LIN {X 0,Y 574.016,Z 518.024,A -85,B 0,C 180,E1 -2272.305,E2 -2272.305} C_VEL
LIN {X 0,Y 573.235,Z 513.083,A -85,B 0,C 180,E1 -2273.099,E2 -2273.099} C_VEL
LIN {X 0,Y 573.254,Z 513.082,A -85,B 0,C 180,E1 -2275.409,E2 -2275.409} C_VEL
LIN {X 0,Y 573.253,Z 513.075,A -85,B 0,C 180,E1 -2278.029,E2 -2278.029} C_VEL
LIN {X 0,Y 573.238,Z 513.077,A -85,B 0,C 180,E1 -2280.883,E2 -2280.883} C_VEL
LIN {X 0,Y 573.261,Z 513.081,A -85,B 0,C 180,E1 -2283.523,E2 -2283.523} C_VEL
LIN {X 0,Y 573.236,Z 513.076,A -85,B 0,C 180,E1 -2286.049,E2 -2286.049} C_VEL
LIN {X 0,Y 573.246,Z 513.073,A -85,B 0,C 180,E1 -2288.7,E2 -2288.7} C_VEL
LIN {X 0,Y 573.251,Z 513.08,A -85,B 0,C 180,E1 -2291.595,E2 -2291.595} C_VEL
LIN {X 0,Y 573.235,Z 513.074,A -85,B 0,C 180,E1 -2294.332,E2 -2294.332} C_VEL
LIN {X 0,Y 573.234,Z 513.083,A -85,B 0,C 180,E1 -2297.358,E2 -2297.358} C_VEL
LIN {X 0,Y 573.243,Z 513.073,A -85,B 0,C 180,E1 -2300.392,E2 -2300.392} C_VEL
LIN {X 0,Y 573.25,Z 513.077,A -85,B 0,C 180,E1 -2303.077,E2 -2303.077} C_VEL
LIN {X 0,Y 573.269,Z 513.077,A -85,B 0,C 180,E1 -2305.671,E2 -2305.671} C_VEL
LIN {X 0,Y 573.243,Z 513.074,A -85,B 0,C 180,E1 -2308.185,E2 -2308.185} C_VEL
LIN {X 0,Y 573.263,Z 513.071,A -85,B 0,C 180,E1 -2310.634,E2 -2310.634} C_VEL
LIN {X 0,Y 573.262,Z 513.081,A -85,B 0,C 180,E1 -2313.5,E2 -2313.5} C_VEL
LIN {X 0,Y 573.224,Z 513.077,A -85,B 0,C 180,E1 -2316.134,E2 -2316.134} C_VEL
LIN {X 0,Y 573.253,Z 513.078,A -85,B 0,C 180,E1 -2319.174,E2 -2319.174} C_VEL
LIN {X 0,Y 573.232,Z 513.085,A -85,B 0,C 180,E1 -2321.412,E2 -2321.412} C_VEL
LIN {X 0,Y 573.249,Z 513.08,A -85,B 0,C 180,E1 -2323.622,E2 -2323.622} C_VEL
LIN {X 0,Y 573.227,Z 513.075,A -85,B 0,C 180,E1 -2326.529,E2 -2326.529} C_VEL
LIN {X 0,Y 573.273,Z 513.07,A -85,B 0,C 180,E1 -2328.734,E2 -2328.734} C_VEL
LIN {X 0,Y 573.298,Z 513.075,A -85,B 0,C 180,E1 -2331.541,E2 -2331.541} C_VEL
LIN {X 0,Y 573.283,Z 513.068,A -85,B 0,C 180,E1 -2334.372,E2 -2334.372} C_VEL
LIN {X 0,Y 573.3,Z 513.069,A -85,B 0,C 180,E1 -2337.892,E2 -2337.892} C_VEL
LIN {X 0,Y 573.328,Z 513.063,A -85,B 0,C 180,E1 -2340.702,E2 -2340.702} C_VEL
LIN {X 0,Y 573.234,Z 513.083,A -85,B 0,C 180,E1 -2343.515,E2 -2343.515} C_VEL
LIN {X 0,Y 573.283,Z 513.075,A -85,B 0,C 180,E1 -2345.628,E2 -2345.628} C_VEL
LIN {X 0,Y 573.298,Z 513.066,A -85,B 0,C 180,E1 -2348.459,E2 -2348.459} C_VEL
LIN {X 0,Y 573.289,Z 513.076,A -85,B 0,C 180,E1 -2351.312,E2 -2351.312} C_VEL
LIN {X 0,Y 573.271,Z 513.07,A -85,B 0,C 180,E1 -2354.425,E2 -2354.425} C_VEL
LIN {X 0,Y 573.25,Z 513.077,A -85,B 0,C 180,E1 -2357.112,E2 -2357.112} C_VEL
LIN {X 0,Y 573.248,Z 513.074,A -85,B 0,C 180,E1 -2360.077,E2 -2360.077} C_VEL
LIN {X 0,Y 573.231,Z 513.075,A -85,B 0,C 180,E1 -2362.338,E2 -2362.338} C_VEL
LIN {X 0,Y 573.243,Z 513.073,A -85,B 0,C 180,E1 -2364.401,E2 -2364.401} C_VEL
LIN {X 0,Y 572.618,Z 513.155,A -85,B 0,C 180,E1 -2364.987,E2 -2364.987} C_VEL
LIN {X 0,Y 569.781,Z 513.514,A -85,B 0,C 180,E1 -2365.939,E2 -2365.939} C_VEL
LIN {X 0,Y 567.353,Z 513.82,A -85,B 0,C 180,E1 -2366.705,E2 -2366.705} C_VEL
LIN {X 0,Y 566.3,Z 513.947,A -85,B 0,C 180,E1 -2367.296,E2 -2367.296} C_VEL
LIN {X 0,Y 566.211,Z 513.956,A -85,B 0,C 180,E1 -2367.496,E2 -2367.496} C_VEL
LIN {X 0,Y 566.221,Z 513.953,A -85,B 0,C 180,E1 -2369.768,E2 -2369.768} C_VEL
LIN {X 0,Y 566.202,Z 513.95,A -85,B 0,C 180,E1 -2372.432,E2 -2372.432} C_VEL
LIN {X 0,Y 566.21,Z 513.953,A -85,B 0,C 180,E1 -2374.996,E2 -2374.996} C_VEL
LIN {X 0,Y 566.191,Z 513.961,A -85,B 0,C 180,E1 -2377.462,E2 -2377.462} C_VEL
LIN {X 0,Y 566.222,Z 513.948,A -85,B 0,C 180,E1 -2380.198,E2 -2380.198} C_VEL
LIN {X 0,Y 566.197,Z 513.956,A -85,B 0,C 180,E1 -2383.055,E2 -2383.055} C_VEL
LIN {X 0,Y 566.2,Z 513.952,A -85,B 0,C 180,E1 -2386.049,E2 -2386.049} C_VEL
LIN {X 0,Y 566.21,Z 513.952,A -85,B 0,C 180,E1 -2388.865,E2 -2388.865} C_VEL
LIN {X 0,Y 566.189,Z 513.958,A -85,B 0,C 180,E1 -2391.638,E2 -2391.638} C_VEL
LIN {X 0,Y 566.193,Z 513.952,A -85,B 0,C 180,E1 -2394.311,E2 -2394.311} C_VEL
LIN {X 0,Y 566.22,Z 513.951,A -85,B 0,C 180,E1 -2396.899,E2 -2396.899} C_VEL
LIN {X 0,Y 566.186,Z 513.963,A -85,B 0,C 180,E1 -2399.408,E2 -2399.408} C_VEL
LIN {X 0,Y 566.213,Z 513.952,A -85,B 0,C 180,E1 -2401.858,E2 -2401.858} C_VEL
LIN {X 0,Y 566.215,Z 513.949,A -85,B 0,C 180,E1 -2404.252,E2 -2404.252} C_VEL
LIN {X 0,Y 566.172,Z 513.955,A -85,B 0,C 180,E1 -2406.72,E2 -2406.72} C_VEL
LIN {X 0,Y 566.217,Z 513.956,A -85,B 0,C 180,E1 -2409.663,E2 -2409.663} C_VEL
LIN {X 0,Y 566.204,Z 513.953,A -85,B 0,C 180,E1 -2412.669,E2 -2412.669} C_VEL
LIN {X 0,Y 566.279,Z 514.062,A -85,B 0,C 180,E1 -2414.178,E2 -2414.178} C_VEL
LIN {X 0,Y 566.581,Z 518.022,A -85,B 0,C 180,E1 -2414.901,E2 -2414.901} C_VEL
LIN {X 0,Y 566.388,Z 534.477,A -85,B 0,C 180,E1 -2417.823,E2 -2417.823} C_VEL
LIN {X 0,Y 566.243,Z 547.118,A -85,B 0,C 180,E1 -2420.039,E2 -2420.039} C_VEL
LIN {X 0,Y 567.168,Z 552.643,A -85,B 0,C 180,E1 -2420.145,E2 -2420.145} C_VEL
LIN {X 0,Y 566.949,Z 653.825,A -85,B 0,C 180,E1 -2421.445,E2 -2421.445} C_VEL
LIN {X 0,Y 566.838,Z 667.023,A -85,B 0,C 180,E1 -2421.758,E2 -2421.758} C_VEL
LIN {X 0,Y 566.748,Z 679.661,A -85,B 0,C 180,E1 -2422.205,E2 -2422.205} C_VEL
LIN {X 0,Y 566.617,Z 691.734,A -85,B 0,C 180,E1 -2422.786,E2 -2422.786} C_VEL
LIN {X 0,Y 566.435,Z 703.285,A -85,B 0,C 180,E1 -2423.506,E2 -2423.506} C_VEL
LIN {X 0,Y 566.299,Z 714.55,A -85,B 0,C 180,E1 -2424.392,E2 -2424.392} C_VEL
LIN {X 0,Y 566.217,Z 724.449,A -85,B 0,C 180,E1 -2425.372,E2 -2425.372} C_VEL
LIN {X 0,Y 566.049,Z 733.188,A -85,B 0,C 180,E1 -2426.441,E2 -2426.441} C_VEL
LIN {X 0,Y 566.022,Z 740.193,A -85,B 0,C 180,E1 -2427.509,E2 -2427.509} C_VEL
LIN {X 0,Y 565.892,Z 745.807,A -85,B 0,C 180,E1 -2428.577,E2 -2428.577} C_VEL
LIN {X 0,Y 565.948,Z 750.233,A -85,B 0,C 180,E1 -2429.644,E2 -2429.644} C_VEL
LIN {X 0,Y 565.846,Z 753.603,A -85,B 0,C 180,E1 -2430.712,E2 -2430.712} C_VEL
LIN {X 0,Y 565.847,Z 755.279,A -85,B 0,C 180,E1 -2431.423,E2 -2431.423} C_VEL
LIN {X 0,Y 565.873,Z 757.434,A -85,B 0,C 180,E1 -2432.847,E2 -2432.847} C_VEL
LIN {X 0,Y 565.911,Z 757.899,A -85,B 0,C 180,E1 -2433.56,E2 -2433.56} C_VEL
LIN {X 0,Y 565.911,Z 757.956,A -85,B 0,C 180,E1 -2434.273,E2 -2434.273} C_VEL
LIN {X 0,Y 565.899,Z 756.923,A -85,B 0,C 180,E1 -2435.702,E2 -2435.702} C_VEL
LIN {X 0,Y 565.919,Z 755.545,A -85,B 0,C 180,E1 -2436.534,E2 -2436.534} C_VEL
LIN {X 0,Y 565.903,Z 752.224,A -85,B 0,C 180,E1 -2437.852,E2 -2437.852} C_VEL
LIN {X 0,Y 565.93,Z 748.356,A -85,B 0,C 180,E1 -2438.93,E2 -2438.93} C_VEL
LIN {X 0,Y 565.978,Z 743.338,A -85,B 0,C 180,E1 -2440.011,E2 -2440.011} C_VEL
LIN {X 0,Y 566.048,Z 736.125,A -85,B 0,C 180,E1 -2441.227,E2 -2441.227} C_VEL
LIN {X 0,Y 566.156,Z 727.551,A -85,B 0,C 180,E1 -2442.364,E2 -2442.364} C_VEL
LIN {X 0,Y 566.247,Z 719.111,A -85,B 0,C 180,E1 -2443.274,E2 -2443.274} C_VEL
LIN {X 0,Y 566.393,Z 708.668,A -85,B 0,C 180,E1 -2444.185,E2 -2444.185} C_VEL
LIN {X 0,Y 566.497,Z 697.979,A -85,B 0,C 180,E1 -2444.936,E2 -2444.936} C_VEL
LIN {X 0,Y 566.671,Z 686.887,A -85,B 0,C 180,E1 -2445.557,E2 -2445.557} C_VEL
LIN {X 0,Y 566.777,Z 675.235,A -85,B 0,C 180,E1 -2446.061,E2 -2446.061} C_VEL
LIN {X 0,Y 566.899,Z 662.692,A -85,B 0,C 180,E1 -2446.451,E2 -2446.451} C_VEL
LIN {X 0,Y 566.964,Z 650.026,A -85,B 0,C 180,E1 -2446.704,E2 -2446.704} C_VEL
LIN {X 0,Y 567.069,Z 552.012,A -85,B 0,C 180,E1 -2447.955,E2 -2447.955} C_VEL
LIN {X 0,Y 566.284,Z 547.177,A -85,B 0,C 180,E1 -2448.04,E2 -2448.04} C_VEL
LIN {X 0,Y 566.438,Z 529.829,A -85,B 0,C 180,E1 -2451.088,E2 -2451.088} C_VEL
LIN {X 0,Y 566.502,Z 515.841,A -85,B 0,C 180,E1 -2453.583,E2 -2453.583} C_VEL
LIN {X 0,Y 566.223,Z 513.955,A -85,B 0,C 180,E1 -2453.936,E2 -2453.936} C_VEL
LIN {X 0,Y 566.21,Z 513.96,A -85,B 0,C 180,E1 -2456.659,E2 -2456.659} C_VEL
LIN {X 0,Y 566.194,Z 513.959,A -85,B 0,C 180,E1 -2458.952,E2 -2458.952} C_VEL
LIN {X 0,Y 566.198,Z 513.952,A -85,B 0,C 180,E1 -2461.421,E2 -2461.421} C_VEL
LIN {X 0,Y 566.21,Z 513.951,A -85,B 0,C 180,E1 -2463.955,E2 -2463.955} C_VEL
LIN {X 0,Y 566.211,Z 513.958,A -85,B 0,C 180,E1 -2466.568,E2 -2466.568} C_VEL
LIN {X 0,Y 566.211,Z 513.95,A -85,B 0,C 180,E1 -2469.685,E2 -2469.685} C_VEL
LIN {X 0,Y 566.214,Z 513.951,A -85,B 0,C 180,E1 -2472.086,E2 -2472.086} C_VEL
LIN {X 0,Y 566.17,Z 513.959,A -85,B 0,C 180,E1 -2475.035,E2 -2475.035} C_VEL
LIN {X 0,Y 566.214,Z 513.951,A -85,B 0,C 180,E1 -2478.135,E2 -2478.135} C_VEL
LIN {X 0,Y 566.217,Z 513.958,A -85,B 0,C 180,E1 -2480.726,E2 -2480.726} C_VEL
LIN {X 0,Y 566.213,Z 513.949,A -85,B 0,C 180,E1 -2483.782,E2 -2483.782} C_VEL
LIN {X 0,Y 566.223,Z 513.952,A -85,B 0,C 180,E1 -2486.262,E2 -2486.262} C_VEL
LIN {X 0,Y 566.196,Z 513.956,A -85,B 0,C 180,E1 -2488.921,E2 -2488.921} C_VEL
LIN {X 0,Y 566.19,Z 513.956,A -85,B 0,C 180,E1 -2491.046,E2 -2491.046} C_VEL
LIN {X 0,Y 566.238,Z 513.945,A -85,B 0,C 180,E1 -2493.46,E2 -2493.46} C_VEL
LIN {X 0,Y 566.191,Z 513.952,A -85,B 0,C 180,E1 -2495.819,E2 -2495.819} C_VEL
LIN {X 0,Y 566.209,Z 513.956,A -85,B 0,C 180,E1 -2498.902,E2 -2498.902} C_VEL
LIN {X 0,Y 566.205,Z 513.952,A -85,B 0,C 180,E1 -2501.172,E2 -2501.172} C_VEL
LIN {X 0,Y 566.212,Z 513.95,A -85,B 0,C 180,E1 -2503.412,E2 -2503.412} C_VEL
LIN {X 0,Y 566.191,Z 513.957,A -85,B 0,C 180,E1 -2506.359,E2 -2506.359} C_VEL
LIN {X 0,Y 566.265,Z 513.953,A -85,B 0,C 180,E1 -2508.654,E2 -2508.654} C_VEL
LIN {X 0,Y 566.239,Z 513.946,A -85,B 0,C 180,E1 -2511.434,E2 -2511.434} C_VEL
LIN {X 0,Y 566.252,Z 513.949,A -85,B 0,C 180,E1 -2514.302,E2 -2514.302} C_VEL
LIN {X 0,Y 566.272,Z 513.941,A -85,B 0,C 180,E1 -2517.866,E2 -2517.866} C_VEL
LIN {X 0,Y 566.298,Z 513.947,A -85,B 0,C 180,E1 -2520.711,E2 -2520.711} C_VEL
LIN {X 0,Y 566.272,Z 513.947,A -85,B 0,C 180,E1 -2522.845,E2 -2522.845} C_VEL
LIN {X 0,Y 566.252,Z 513.945,A -85,B 0,C 180,E1 -2525.698,E2 -2525.698} C_VEL
LIN {X 0,Y 566.24,Z 513.955,A -85,B 0,C 180,E1 -2528.565,E2 -2528.565} C_VEL
LIN {X 0,Y 566.241,Z 513.946,A -85,B 0,C 180,E1 -2531.454,E2 -2531.454} C_VEL
LIN {X 0,Y 566.223,Z 513.955,A -85,B 0,C 180,E1 -2534.507,E2 -2534.507} C_VEL
LIN {X 0,Y 566.194,Z 513.952,A -85,B 0,C 180,E1 -2537.332,E2 -2537.332} C_VEL
LIN {X 0,Y 566.211,Z 513.955,A -85,B 0,C 180,E1 -2540.337,E2 -2540.337} C_VEL
LIN {X 0,Y 566.18,Z 513.953,A -85,B 0,C 180,E1 -2543.404,E2 -2543.404} C_VEL
LIN {X 0,Y 566.218,Z 513.949,A -85,B 0,C 180,E1 -2545.749,E2 -2545.749} C_VEL
LIN {X 0,Y 566.199,Z 513.954,A -85,B 0,C 180,E1 -2548.204,E2 -2548.204} C_VEL
LIN {X 0,Y 566.187,Z 513.963,A -85,B 0,C 180,E1 -2550.592,E2 -2550.592} C_VEL
LIN {X 0,Y 566.222,Z 513.95,A -85,B 0,C 180,E1 -2553.102,E2 -2553.102} C_VEL
LIN {X 0,Y 566.207,Z 513.95,A -85,B 0,C 180,E1 -2555.689,E2 -2555.689} C_VEL
LIN {X 0,Y 566.21,Z 513.96,A -85,B 0,C 180,E1 -2558.56,E2 -2558.56} C_VEL
LIN {X 0,Y 566.206,Z 513.952,A -85,B 0,C 180,E1 -2561.137,E2 -2561.137} C_VEL
LIN {X 0,Y 566.192,Z 513.955,A -85,B 0,C 180,E1 -2564.036,E2 -2564.036} C_VEL
LIN {X 0,Y 566.201,Z 513.953,A -85,B 0,C 180,E1 -2567.083,E2 -2567.083} C_VEL
LIN {X 0,Y 566.224,Z 513.949,A -85,B 0,C 180,E1 -2569.804,E2 -2569.804} C_VEL
LIN {X 0,Y 566.196,Z 513.961,A -85,B 0,C 180,E1 -2572.6,E2 -2572.6} C_VEL
LIN {X 0,Y 566.206,Z 513.952,A -85,B 0,C 180,E1 -2575.183,E2 -2575.183} C_VEL
LIN {X 0,Y 566.233,Z 513.948,A -85,B 0,C 180,E1 -2577.744,E2 -2577.744} C_VEL
LIN {X 0,Y 566.203,Z 513.958,A -85,B 0,C 180,E1 -2580.328,E2 -2580.328} C_VEL
LIN {X 0,Y 566.212,Z 513.959,A -85,B 0,C 180,E1 -2582.662,E2 -2582.662} C_VEL
LIN {X 0,Y 566.237,Z 513.952,A -85,B 0,C 180,E1 -2585.04,E2 -2585.04} C_VEL
LIN {X 0,Y 566.184,Z 514.02,A -85,B 0,C 180,E1 -2586.755,E2 -2586.755} C_VEL
LIN {X 0,Y 567.094,Z 519.284,A -85,B 0,C 180,E1 -2587.6,E2 -2587.6} C_VEL
LIN {X 0,Y 566.787,Z 539.05,A -85,B 0,C 180,E1 -2590.572,E2 -2590.572} C_VEL
LIN {X 0,Y 566.56,Z 557.206,A -85,B 0,C 180,E1 -2593.259,E2 -2593.259} C_VEL
LIN {X 0,Y 566.392,Z 576.169,A -85,B 0,C 180,E1 -2595.998,E2 -2595.998} C_VEL
LIN {X 0,Y 567.213,Z 582.317,A -85,B 0,C 180,E1 -2596.097,E2 -2596.097} C_VEL
LIN {X 0,Y 566.955,Z 683.962,A -85,B 0,C 180,E1 -2597.403,E2 -2597.403} C_VEL
LIN {X 0,Y 566.847,Z 697.229,A -85,B 0,C 180,E1 -2597.719,E2 -2597.719} C_VEL
LIN {X 0,Y 566.758,Z 709.382,A -85,B 0,C 180,E1 -2598.149,E2 -2598.149} C_VEL
LIN {X 0,Y 566.627,Z 721.158,A -85,B 0,C 180,E1 -2598.708,E2 -2598.708} C_VEL
LIN {X 0,Y 566.457,Z 733.205,A -85,B 0,C 180,E1 -2599.456,E2 -2599.456} C_VEL
LIN {X 0,Y 566.318,Z 743.604,A -85,B 0,C 180,E1 -2600.266,E2 -2600.266} C_VEL
LIN {X 0,Y 566.207,Z 752.115,A -85,B 0,C 180,E1 -2601.074,E2 -2601.074} C_VEL
LIN {X 0,Y 566.112,Z 759.962,A -85,B 0,C 180,E1 -2601.972,E2 -2601.972} C_VEL
LIN {X 0,Y 566.003,Z 767.623,A -85,B 0,C 180,E1 -2603.047,E2 -2603.047} C_VEL
LIN {X 0,Y 566.004,Z 774.681,A -85,B 0,C 180,E1 -2604.299,E2 -2604.299} C_VEL
LIN {X 0,Y 565.933,Z 779.372,A -85,B 0,C 180,E1 -2605.37,E2 -2605.37} C_VEL
LIN {X 0,Y 565.927,Z 782.958,A -85,B 0,C 180,E1 -2606.44,E2 -2606.44} C_VEL
LIN {X 0,Y 565.878,Z 784.808,A -85,B 0,C 180,E1 -2607.153,E2 -2607.153} C_VEL
LIN {X 0,Y 565.846,Z 787.186,A -85,B 0,C 180,E1 -2608.577,E2 -2608.577} C_VEL
LIN {X 0,Y 565.839,Z 788,A -85,B 0,C 180,E1 -2610,E2 -2610} C_VEL
LIN {X 0,Y 565.846,Z 787.186,A -85,B 0,C 180,E1 -2611.423,E2 -2611.423} C_VEL
LIN {X 0,Y 565.878,Z 784.81,A -85,B 0,C 180,E1 -2612.847,E2 -2612.847} C_VEL
LIN {X 0,Y 565.926,Z 781.896,A -85,B 0,C 180,E1 -2613.916,E2 -2613.916} C_VEL
LIN {X 0,Y 565.878,Z 777.949,A -85,B 0,C 180,E1 -2614.987,E2 -2614.987} C_VEL
LIN {X 0,Y 566.002,Z 772.867,A -85,B 0,C 180,E1 -2616.058,E2 -2616.058} C_VEL
LIN {X 0,Y 566.04,Z 766.47,A -85,B 0,C 180,E1 -2617.132,E2 -2617.132} C_VEL
LIN {X 0,Y 566.133,Z 758.48,A -85,B 0,C 180,E1 -2618.207,E2 -2618.207} C_VEL
LIN {X 0,Y 566.228,Z 750.338,A -85,B 0,C 180,E1 -2619.105,E2 -2619.105} C_VEL
LIN {X 0,Y 566.341,Z 740.404,A -85,B 0,C 180,E1 -2620.005,E2 -2620.005} C_VEL
LIN {X 0,Y 566.523,Z 729.288,A -85,B 0,C 180,E1 -2620.808,E2 -2620.808} C_VEL
LIN {X 0,Y 566.66,Z 718.182,A -85,B 0,C 180,E1 -2621.445,E2 -2621.445} C_VEL
LIN {X 0,Y 566.74,Z 705.991,A -85,B 0,C 180,E1 -2621.988,E2 -2621.988} C_VEL
LIN {X 0,Y 566.881,Z 693.188,A -85,B 0,C 180,E1 -2622.394,E2 -2622.394} C_VEL
LIN {X 0,Y 567.009,Z 679.622,A -85,B 0,C 180,E1 -2622.664,E2 -2622.664} C_VEL
LIN {X 0,Y 567.037,Z 580.204,A -85,B 0,C 180,E1 -2623.934,E2 -2623.934} C_VEL
LIN {X 0,Y 566.374,Z 575.795,A -85,B 0,C 180,E1 -2624.025,E2 -2624.025} C_VEL
LIN {X 0,Y 566.57,Z 556.089,A -85,B 0,C 180,E1 -2626.906,E2 -2626.906} C_VEL
LIN {X 0,Y 566.777,Z 538.173,A -85,B 0,C 180,E1 -2629.56,E2 -2629.56} C_VEL
LIN {X 0,Y 567.094,Z 519.284,A -85,B 0,C 180,E1 -2632.4,E2 -2632.4} C_VEL
LIN {X 0,Y 566.19,Z 513.961,A -85,B 0,C 180,E1 -2633.285,E2 -2633.285} C_VEL
LIN {X 0,Y 566.213,Z 513.956,A -85,B 0,C 180,E1 -2635.748,E2 -2635.748} C_VEL
LIN {X 0,Y 566.202,Z 513.952,A -85,B 0,C 180,E1 -2638.201,E2 -2638.201} C_VEL
LIN {X 0,Y 566.199,Z 513.956,A -85,B 0,C 180,E1 -2641.077,E2 -2641.077} C_VEL
LIN {X 0,Y 566.21,Z 513.955,A -85,B 0,C 180,E1 -2643.733,E2 -2643.733} C_VEL
LIN {X 0,Y 566.205,Z 513.95,A -85,B 0,C 180,E1 -2646.568,E2 -2646.568} C_VEL
LIN {X 0,Y 566.21,Z 513.956,A -85,B 0,C 180,E1 -2649.685,E2 -2649.685} C_VEL
LIN {X 0,Y 566.211,Z 513.951,A -85,B 0,C 180,E1 -2652.086,E2 -2652.086} C_VEL
LIN {X 0,Y 566.168,Z 513.958,A -85,B 0,C 180,E1 -2655.035,E2 -2655.035} C_VEL
LIN {X 0,Y 566.212,Z 513.95,A -85,B 0,C 180,E1 -2658.135,E2 -2658.135} C_VEL
LIN {X 0,Y 566.217,Z 513.949,A -85,B 0,C 180,E1 -2660.726,E2 -2660.726} C_VEL
LIN {X 0,Y 566.212,Z 513.954,A -85,B 0,C 180,E1 -2663.783,E2 -2663.783} C_VEL
LIN {X 0,Y 566.222,Z 513.948,A -85,B 0,C 180,E1 -2666.262,E2 -2666.262} C_VEL
LIN {X 0,Y 566.195,Z 513.954,A -85,B 0,C 180,E1 -2668.921,E2 -2668.921} C_VEL
LIN {X 0,Y 566.19,Z 513.956,A -85,B 0,C 180,E1 -2671.046,E2 -2671.046} C_VEL
LIN {X 0,Y 566.237,Z 513.957,A -85,B 0,C 180,E1 -2673.46,E2 -2673.46} C_VEL
LIN {X 0,Y 566.19,Z 513.956,A -85,B 0,C 180,E1 -2675.819,E2 -2675.819} C_VEL
LIN {X 0,Y 566.208,Z 513.952,A -85,B 0,C 180,E1 -2678.902,E2 -2678.902} C_VEL
LIN {X 0,Y 566.205,Z 513.956,A -85,B 0,C 180,E1 -2681.172,E2 -2681.172} C_VEL
LIN {X 0,Y 566.211,Z 513.959,A -85,B 0,C 180,E1 -2683.412,E2 -2683.412} C_VEL
LIN {X 0,Y 566.189,Z 513.952,A -85,B 0,C 180,E1 -2686.359,E2 -2686.359} C_VEL
LIN {X 0,Y 566.265,Z 513.943,A -85,B 0,C 180,E1 -2688.654,E2 -2688.654} C_VEL
LIN {X 0,Y 566.239,Z 513.956,A -85,B 0,C 180,E1 -2691.435,E2 -2691.435} C_VEL
LIN {X 0,Y 566.251,Z 513.944,A -85,B 0,C 180,E1 -2694.302,E2 -2694.302} C_VEL
LIN {X 0,Y 566.271,Z 513.945,A -85,B 0,C 180,E1 -2697.866,E2 -2697.866} C_VEL
LIN {X 0,Y 566.298,Z 513.939,A -85,B 0,C 180,E1 -2700.711,E2 -2700.711} C_VEL
LIN {X 0,Y 566.271,Z 513.944,A -85,B 0,C 180,E1 -2702.846,E2 -2702.846} C_VEL
LIN {X 0,Y 566.251,Z 513.95,A -85,B 0,C 180,E1 -2705.698,E2 -2705.698} C_VEL
LIN {X 0,Y 566.239,Z 513.946,A -85,B 0,C 180,E1 -2708.566,E2 -2708.566} C_VEL
LIN {X 0,Y 566.241,Z 513.956,A -85,B 0,C 180,E1 -2711.454,E2 -2711.454} C_VEL
LIN {X 0,Y 566.224,Z 513.948,A -85,B 0,C 180,E1 -2714.507,E2 -2714.507} C_VEL
LIN {X 0,Y 566.195,Z 513.96,A -85,B 0,C 180,E1 -2717.332,E2 -2717.332} C_VEL
LIN {X 0,Y 566.211,Z 513.949,A -85,B 0,C 180,E1 -2720.337,E2 -2720.337} C_VEL
LIN {X 0,Y 566.181,Z 513.963,A -85,B 0,C 180,E1 -2723.404,E2 -2723.404} C_VEL
LIN {X 0,Y 566.219,Z 513.953,A -85,B 0,C 180,E1 -2725.749,E2 -2725.749} C_VEL
LIN {X 0,Y 566.211,Z 513.956,A -85,B 0,C 180,E1 -2727.496,E2 -2727.496} C_VEL
LIN {X 0,Y 565.532,Z 514.036,A -85,B 0,C 180,E1 -2728.09,E2 -2728.09} C_VEL
LIN {X 0,Y 562.667,Z 514.395,A -85,B 0,C 180,E1 -2729.054,E2 -2729.054} C_VEL
LIN {X 0,Y 560.256,Z 514.695,A -85,B 0,C 180,E1 -2729.829,E2 -2729.829} C_VEL
LIN {X 0,Y 559.227,Z 514.82,A -85,B 0,C 180,E1 -2730.428,E2 -2730.428} C_VEL
LIN {X 0,Y 559.146,Z 514.83,A -85,B 0,C 180,E1 -2730.631,E2 -2730.631} C_VEL
LIN {X 0,Y 559.172,Z 514.833,A -85,B 0,C 180,E1 -2733.575,E2 -2733.575} C_VEL
LIN {X 0,Y 559.164,Z 514.827,A -85,B 0,C 180,E1 -2736.449,E2 -2736.449} C_VEL
LIN {X 0,Y 559.173,Z 514.829,A -85,B 0,C 180,E1 -2738.935,E2 -2738.935} C_VEL
LIN {X 0,Y 559.187,Z 514.828,A -85,B 0,C 180,E1 -2741.768,E2 -2741.768} C_VEL
LIN {X 0,Y 559.136,Z 514.832,A -85,B 0,C 180,E1 -2744.74,E2 -2744.74} C_VEL
LIN {X 0,Y 559.165,Z 514.835,A -85,B 0,C 180,E1 -2747.258,E2 -2747.258} C_VEL
LIN {X 0,Y 559.184,Z 514.825,A -85,B 0,C 180,E1 -2750.136,E2 -2750.136} C_VEL
LIN {X 0,Y 559.144,Z 514.832,A -85,B 0,C 180,E1 -2752.893,E2 -2752.893} C_VEL
LIN {X 0,Y 559.166,Z 514.828,A -85,B 0,C 180,E1 -2756.052,E2 -2756.052} C_VEL
LIN {X 0,Y 559.16,Z 514.831,A -85,B 0,C 180,E1 -2758.982,E2 -2758.982} C_VEL
LIN {X 0,Y 559.169,Z 514.833,A -85,B 0,C 180,E1 -2761.62,E2 -2761.62} C_VEL
LIN {X 0,Y 559.182,Z 514.827,A -85,B 0,C 180,E1 -2763.904,E2 -2763.904} C_VEL
LIN {X 0,Y 559.142,Z 514.83,A -85,B 0,C 180,E1 -2766.572,E2 -2766.572} C_VEL
LIN {X 0,Y 559.183,Z 514.836,A -85,B 0,C 180,E1 -2769.396,E2 -2769.396} C_VEL
LIN {X 0,Y 559.151,Z 514.837,A -85,B 0,C 180,E1 -2771.686,E2 -2771.686} C_VEL
LIN {X 0,Y 559.236,Z 515.011,A -85,B 0,C 180,E1 -2774.091,E2 -2774.091} C_VEL
LIN {X 0,Y 559.619,Z 518.326,A -85,B 0,C 180,E1 -2774.709,E2 -2774.709} C_VEL
LIN {X 0,Y 559.362,Z 535.81,A -85,B 0,C 180,E1 -2777.851,E2 -2777.851} C_VEL
LIN {X 0,Y 559.198,Z 547.161,A -85,B 0,C 180,E1 -2779.866,E2 -2779.866} C_VEL
LIN {X 0,Y 560.281,Z 554.897,A -85,B 0,C 180,E1 -2780,E2 -2780} C_VEL
LIN {X 0,Y 560.036,Z 654.138,A -85,B 0,C 180,E1 -2781.294,E2 -2781.294} C_VEL
LIN {X 0,Y 559.908,Z 667.231,A -85,B 0,C 180,E1 -2781.61,E2 -2781.61} C_VEL
LIN {X 0,Y 559.779,Z 679.821,A -85,B 0,C 180,E1 -2782.062,E2 -2782.062} C_VEL
LIN {X 0,Y 559.657,Z 691.048,A -85,B 0,C 180,E1 -2782.605,E2 -2782.605} C_VEL
LIN {X 0,Y 559.465,Z 702.826,A -85,B 0,C 180,E1 -2783.34,E2 -2783.34} C_VEL
LIN {X 0,Y 559.31,Z 714.108,A -85,B 0,C 180,E1 -2784.231,E2 -2784.231} C_VEL
LIN {X 0,Y 559.221,Z 723.294,A -85,B 0,C 180,E1 -2785.134,E2 -2785.134} C_VEL
LIN {X 0,Y 559.062,Z 732.224,A -85,B 0,C 180,E1 -2786.216,E2 -2786.216} C_VEL
LIN {X 0,Y 558.925,Z 739.434,A -85,B 0,C 180,E1 -2787.297,E2 -2787.297} C_VEL
LIN {X 0,Y 558.88,Z 744.316,A -85,B 0,C 180,E1 -2788.198,E2 -2788.198} C_VEL
LIN {X 0,Y 558.769,Z 749.072,A -85,B 0,C 180,E1 -2789.279,E2 -2789.279} C_VEL
LIN {X 0,Y 558.828,Z 752.727,A -85,B 0,C 180,E1 -2790.36,E2 -2790.36} C_VEL
LIN {X 0,Y 558.746,Z 755.382,A -85,B 0,C 180,E1 -2791.441,E2 -2791.441} C_VEL
LIN {X 0,Y 558.794,Z 757.486,A -85,B 0,C 180,E1 -2792.884,E2 -2792.884} C_VEL
LIN {X 0,Y 558.82,Z 757.91,A -85,B 0,C 180,E1 -2793.605,E2 -2793.605} C_VEL
LIN {X 0,Y 558.762,Z 757.597,A -85,B 0,C 180,E1 -2795.051,E2 -2795.051} C_VEL
LIN {X 0,Y 558.81,Z 756.859,A -85,B 0,C 180,E1 -2795.774,E2 -2795.774} C_VEL
LIN {X 0,Y 558.847,Z 755.605,A -85,B 0,C 180,E1 -2796.535,E2 -2796.535} C_VEL
LIN {X 0,Y 558.83,Z 752.071,A -85,B 0,C 180,E1 -2797.952,E2 -2797.952} C_VEL
LIN {X 0,Y 558.834,Z 748.151,A -85,B 0,C 180,E1 -2799.044,E2 -2799.044} C_VEL
LIN {X 0,Y 558.911,Z 743.077,A -85,B 0,C 180,E1 -2800.139,E2 -2800.139} C_VEL
LIN {X 0,Y 558.982,Z 736.397,A -85,B 0,C 180,E1 -2801.278,E2 -2801.278} C_VEL
LIN {X 0,Y 559.073,Z 728.624,A -85,B 0,C 180,E1 -2802.339,E2 -2802.339} C_VEL
LIN {X 0,Y 559.201,Z 720.399,A -85,B 0,C 180,E1 -2803.259,E2 -2803.259} C_VEL
LIN {X 0,Y 559.356,Z 710.333,A -85,B 0,C 180,E1 -2804.182,E2 -2804.182} C_VEL
LIN {X 0,Y 559.487,Z 699.332,A -85,B 0,C 180,E1 -2804.987,E2 -2804.987} C_VEL
LIN {X 0,Y 559.692,Z 687.654,A -85,B 0,C 180,E1 -2805.662,E2 -2805.662} C_VEL
LIN {X 0,Y 559.839,Z 675.058,A -85,B 0,C 180,E1 -2806.219,E2 -2806.219} C_VEL
LIN {X 0,Y 559.983,Z 662.435,A -85,B 0,C 180,E1 -2806.613,E2 -2806.613} C_VEL
LIN {X 0,Y 560.057,Z 650.139,A -85,B 0,C 180,E1 -2806.861,E2 -2806.861} C_VEL
LIN {X 0,Y 560.254,Z 553.25,A -85,B 0,C 180,E1 -2808.112,E2 -2808.112} C_VEL
LIN {X 0,Y 559.263,Z 547.067,A -85,B 0,C 180,E1 -2808.239,E2 -2808.239} C_VEL
LIN {X 0,Y 559.46,Z 529.514,A -85,B 0,C 180,E1 -2811.364,E2 -2811.364} C_VEL
LIN {X 0,Y 559.56,Z 517.539,A -85,B 0,C 180,E1 -2813.526,E2 -2813.526} C_VEL
LIN {X 0,Y 559.201,Z 514.831,A -85,B 0,C 180,E1 -2814.058,E2 -2814.058} C_VEL
LIN {X 0,Y 559.171,Z 514.835,A -85,B 0,C 180,E1 -2816.902,E2 -2816.902} C_VEL
LIN {X 0,Y 559.15,Z 514.831,A -85,B 0,C 180,E1 -2819.857,E2 -2819.857} C_VEL
LIN {X 0,Y 559.174,Z 514.836,A -85,B 0,C 180,E1 -2822.713,E2 -2822.713} C_VEL
LIN {X 0,Y 559.145,Z 514.832,A -85,B 0,C 180,E1 -2825.322,E2 -2825.322} C_VEL
LIN {X 0,Y 559.134,Z 514.832,A -85,B 0,C 180,E1 -2828.016,E2 -2828.016} C_VEL
LIN {X 0,Y 559.174,Z 514.834,A -85,B 0,C 180,E1 -2830.81,E2 -2830.81} C_VEL
LIN {X 0,Y 559.161,Z 514.828,A -85,B 0,C 180,E1 -2833.731,E2 -2833.731} C_VEL
LIN {X 0,Y 559.164,Z 514.835,A -85,B 0,C 180,E1 -2836.8,E2 -2836.8} C_VEL
LIN {X 0,Y 559.172,Z 514.827,A -85,B 0,C 180,E1 -2839.189,E2 -2839.189} C_VEL
LIN {X 0,Y 559.129,Z 514.833,A -85,B 0,C 180,E1 -2841.982,E2 -2841.982} C_VEL
LIN {X 0,Y 559.156,Z 514.836,A -85,B 0,C 180,E1 -2844.782,E2 -2844.782} C_VEL
LIN {X 0,Y 559.168,Z 514.828,A -85,B 0,C 180,E1 -2847.36,E2 -2847.36} C_VEL
LIN {X 0,Y 559.183,Z 514.826,A -85,B 0,C 180,E1 -2850.134,E2 -2850.134} C_VEL
LIN {X 0,Y 559.175,Z 514.827,A -85,B 0,C 180,E1 -2853.169,E2 -2853.169} C_VEL
LIN {X 0,Y 559.149,Z 514.83,A -85,B 0,C 180,E1 -2855.494,E2 -2855.494} C_VEL
LIN {X 0,Y 559.169,Z 514.835,A -85,B 0,C 180,E1 -2858.624,E2 -2858.624} C_VEL
LIN {X 0,Y 559.163,Z 514.832,A -85,B 0,C 180,E1 -2860.926,E2 -2860.926} C_VEL
LIN {X 0,Y 559.162,Z 514.828,A -85,B 0,C 180,E1 -2863.948,E2 -2863.948} C_VEL
LIN {X 0,Y 559.165,Z 514.83,A -85,B 0,C 180,E1 -2866.184,E2 -2866.184} C_VEL
LIN {X 0,Y 559.201,Z 514.825,A -85,B 0,C 180,E1 -2869.133,E2 -2869.133} C_VEL
LIN {X 0,Y 559.204,Z 514.823,A -85,B 0,C 180,E1 -2872.053,E2 -2872.053} C_VEL
LIN {X 0,Y 559.251,Z 514.821,A -85,B 0,C 180,E1 -2874.953,E2 -2874.953} C_VEL
LIN {X 0,Y 559.243,Z 514.816,A -85,B 0,C 180,E1 -2877.839,E2 -2877.839} C_VEL
LIN {X 0,Y 559.267,Z 514.823,A -85,B 0,C 180,E1 -2880.72,E2 -2880.72} C_VEL
LIN {X 0,Y 559.237,Z 514.822,A -85,B 0,C 180,E1 -2882.881,E2 -2882.881} C_VEL
LIN {X 0,Y 559.221,Z 514.821,A -85,B 0,C 180,E1 -2885.77,E2 -2885.77} C_VEL
LIN {X 0,Y 559.194,Z 514.832,A -85,B 0,C 180,E1 -2888.674,E2 -2888.674} C_VEL
LIN {X 0,Y 559.199,Z 514.823,A -85,B 0,C 180,E1 -2891.601,E2 -2891.601} C_VEL
LIN {X 0,Y 559.189,Z 514.833,A -85,B 0,C 180,E1 -2894.596,E2 -2894.596} C_VEL
LIN {X 0,Y 559.154,Z 514.828,A -85,B 0,C 180,E1 -2897.557,E2 -2897.557} C_VEL
LIN {X 0,Y 559.166,Z 514.828,A -85,B 0,C 180,E1 -2899.838,E2 -2899.838} C_VEL
LIN {X 0,Y 559.134,Z 514.834,A -85,B 0,C 180,E1 -2902.153,E2 -2902.153} C_VEL
LIN {X 0,Y 559.171,Z 514.828,A -85,B 0,C 180,E1 -2905.188,E2 -2905.188} C_VEL
LIN {X 0,Y 559.186,Z 514.824,A -85,B 0,C 180,E1 -2907.712,E2 -2907.712} C_VEL
LIN {X 0,Y 559.161,Z 514.832,A -85,B 0,C 180,E1 -2910.182,E2 -2910.182} C_VEL
LIN {X 0,Y 559.168,Z 514.835,A -85,B 0,C 180,E1 -2912.715,E2 -2912.715} C_VEL
LIN {X 0,Y 559.152,Z 514.829,A -85,B 0,C 180,E1 -2915.322,E2 -2915.322} C_VEL
LIN {X 0,Y 559.129,Z 514.834,A -85,B 0,C 180,E1 -2918.018,E2 -2918.018} C_VEL
LIN {X 0,Y 559.171,Z 514.833,A -85,B 0,C 180,E1 -2920.811,E2 -2920.811} C_VEL
LIN {X 0,Y 559.136,Z 514.832,A -85,B 0,C 180,E1 -2923.735,E2 -2923.735} C_VEL
LIN {X 0,Y 559.164,Z 514.834,A -85,B 0,C 180,E1 -2926.802,E2 -2926.802} C_VEL
LIN {X 0,Y 559.174,Z 514.828,A -85,B 0,C 180,E1 -2929.19,E2 -2929.19} C_VEL
LIN {X 0,Y 559.133,Z 514.834,A -85,B 0,C 180,E1 -2931.983,E2 -2931.983} C_VEL
LIN {X 0,Y 559.143,Z 514.836,A -85,B 0,C 180,E1 -2934.786,E2 -2934.786} C_VEL
LIN {X 0,Y 559.173,Z 514.827,A -85,B 0,C 180,E1 -2937.362,E2 -2937.362} C_VEL
LIN {X 0,Y 559.149,Z 514.834,A -85,B 0,C 180,E1 -2940.143,E2 -2940.143} C_VEL
LIN {X 0,Y 559.169,Z 514.831,A -85,B 0,C 180,E1 -2943.098,E2 -2943.098} C_VEL
LIN {X 0,Y 559.158,Z 514.832,A -85,B 0,C 180,E1 -2945.496,E2 -2945.496} C_VEL
LIN {X 0,Y 559.177,Z 514.94,A -85,B 0,C 180,E1 -2946.608,E2 -2946.608} C_VEL
LIN {X 0,Y 560.178,Z 520.514,A -85,B 0,C 180,E1 -2947.502,E2 -2947.502} C_VEL
LIN {X 0,Y 559.826,Z 539.771,A -85,B 0,C 180,E1 -2950.43,E2 -2950.43} C_VEL
LIN {X 0,Y 559.604,Z 556.396,A -85,B 0,C 180,E1 -2952.923,E2 -2952.923} C_VEL
LIN {X 0,Y 559.405,Z 576.169,A -85,B 0,C 180,E1 -2955.819,E2 -2955.819} C_VEL
LIN {X 0,Y 560.32,Z 583.324,A -85,B 0,C 180,E1 -2955.936,E2 -2955.936} C_VEL
LIN {X 0,Y 560.027,Z 683.962,A -85,B 0,C 180,E1 -2957.245,E2 -2957.245} C_VEL
LIN {X 0,Y 559.923,Z 697.228,A -85,B 0,C 180,E1 -2957.565,E2 -2957.565} C_VEL
LIN {X 0,Y 559.811,Z 709.383,A -85,B 0,C 180,E1 -2958,E2 -2958} C_VEL
LIN {X 0,Y 559.668,Z 720.814,A -85,B 0,C 180,E1 -2958.547,E2 -2958.547} C_VEL
LIN {X 0,Y 559.495,Z 731.912,A -85,B 0,C 180,E1 -2959.231,E2 -2959.231} C_VEL
LIN {X 0,Y 559.309,Z 742.543,A -85,B 0,C 180,E1 -2960.051,E2 -2960.051} C_VEL
LIN {X 0,Y 559.161,Z 752.115,A -85,B 0,C 180,E1 -2960.961,E2 -2960.961} C_VEL
LIN {X 0,Y 559.05,Z 759.962,A -85,B 0,C 180,E1 -2961.87,E2 -2961.87} C_VEL
LIN {X 0,Y 558.943,Z 767.623,A -85,B 0,C 180,E1 -2962.959,E2 -2962.959} C_VEL
LIN {X 0,Y 558.935,Z 774.68,A -85,B 0,C 180,E1 -2964.227,E2 -2964.227} C_VEL
LIN {X 0,Y 558.827,Z 779.373,A -85,B 0,C 180,E1 -2965.311,E2 -2965.311} C_VEL
LIN {X 0,Y 558.836,Z 782.958,A -85,B 0,C 180,E1 -2966.395,E2 -2966.395} C_VEL
LIN {X 0,Y 558.799,Z 784.808,A -85,B 0,C 180,E1 -2967.116,E2 -2967.116} C_VEL
LIN {X 0,Y 558.745,Z 787.185,A -85,B 0,C 180,E1 -2968.559,E2 -2968.559} C_VEL
LIN {X 0,Y 558.74,Z 788,A -85,B 0,C 180,E1 -2970,E2 -2970} C_VEL
LIN {X 0,Y 558.745,Z 787.186,A -85,B 0,C 180,E1 -2971.441,E2 -2971.441} C_VEL
LIN {X 0,Y 558.799,Z 784.81,A -85,B 0,C 180,E1 -2972.884,E2 -2972.884} C_VEL
LIN {X 0,Y 558.843,Z 781.896,A -85,B 0,C 180,E1 -2973.966,E2 -2973.966} C_VEL
LIN {X 0,Y 558.799,Z 777.949,A -85,B 0,C 180,E1 -2975.051,E2 -2975.051} C_VEL
LIN {X 0,Y 558.921,Z 772.868,A -85,B 0,C 180,E1 -2976.135,E2 -2976.135} C_VEL
LIN {X 0,Y 558.977,Z 766.469,A -85,B 0,C 180,E1 -2977.223,E2 -2977.223} C_VEL
LIN {X 0,Y 559.098,Z 758.48,A -85,B 0,C 180,E1 -2978.311,E2 -2978.311} C_VEL
LIN {X 0,Y 559.184,Z 750.337,A -85,B 0,C 180,E1 -2979.221,E2 -2979.221} C_VEL
LIN {X 0,Y 559.352,Z 740.403,A -85,B 0,C 180,E1 -2980.131,E2 -2980.131} C_VEL
LIN {X 0,Y 559.544,Z 729.368,A -85,B 0,C 180,E1 -2980.939,E2 -2980.939} C_VEL
LIN {X 0,Y 559.703,Z 717.148,A -85,B 0,C 180,E1 -2981.643,E2 -2981.643} C_VEL
LIN {X 0,Y 559.819,Z 704.776,A -85,B 0,C 180,E1 -2982.184,E2 -2982.184} C_VEL
LIN {X 0,Y 559.946,Z 691.359,A -85,B 0,C 180,E1 -2982.596,E2 -2982.596} C_VEL
LIN {X 0,Y 560.068,Z 678.106,A -85,B 0,C 180,E1 -2982.846,E2 -2982.846} C_VEL
LIN {X 0,Y 560.194,Z 581.19,A -85,B 0,C 180,E1 -2984.095,E2 -2984.095} C_VEL
LIN {X 0,Y 559.37,Z 575.795,A -85,B 0,C 180,E1 -2984.205,E2 -2984.205} C_VEL
LIN {X 0,Y 559.624,Z 554.49,A -85,B 0,C 180,E1 -2987.361,E2 -2987.361} C_VEL
LIN {X 0,Y 559.94,Z 534.395,A -85,B 0,C 180,E1 -2990.383,E2 -2990.383} C_VEL
LIN {X 0,Y 560.178,Z 520.515,A -85,B 0,C 180,E1 -2992.498,E2 -2992.498} C_VEL
LIN {X 0,Y 559.174,Z 514.835,A -85,B 0,C 180,E1 -2993.436,E2 -2993.436} C_VEL
LIN {X 0,Y 559.181,Z 514.828,A -85,B 0,C 180,E1 -2996.096,E2 -2996.096} C_VEL
LIN {X 0,Y 559.163,Z 514.829,A -85,B 0,C 180,E1 -2998.529,E2 -2998.529} C_VEL
LIN {X 0,Y 559.153,Z 514.837,A -85,B 0,C 180,E1 -3001.274,E2 -3001.274} C_VEL
LIN {X 0,Y 559.164,Z 514.83,A -85,B 0,C 180,E1 -3003.948,E2 -3003.948} C_VEL
LIN {X 0,Y 559.141,Z 514.834,A -85,B 0,C 180,E1 -3007.107,E2 -3007.107} C_VEL
LIN {X 0,Y 559.166,Z 514.83,A -85,B 0,C 180,E1 -3009.942,E2 -3009.942} C_VEL
LIN {X 0,Y 559.16,Z 514.828,A -85,B 0,C 180,E1 -3012.742,E2 -3012.742} C_VEL
LIN {X 0,Y 559.148,Z 514.834,A -85,B 0,C 180,E1 -3015.76,E2 -3015.76} C_VEL
LIN {X 0,Y 559.186,Z 514.825,A -85,B 0,C 180,E1 -3018.232,E2 -3018.232} C_VEL
LIN {X 0,Y 559.172,Z 514.832,A -85,B 0,C 180,E1 -3021.19,E2 -3021.19} C_VEL
LIN {X 0,Y 559.166,Z 514.832,A -85,B 0,C 180,E1 -3023.791,E2 -3023.791} C_VEL
LIN {X 0,Y 559.171,Z 514.826,A -85,B 0,C 180,E1 -3026.426,E2 -3026.426} C_VEL
LIN {X 0,Y 559.159,Z 514.831,A -85,B 0,C 180,E1 -3028.981,E2 -3028.981} C_VEL
LIN {X 0,Y 559.163,Z 514.835,A -85,B 0,C 180,E1 -3031.617,E2 -3031.617} C_VEL
LIN {X 0,Y 559.191,Z 514.827,A -85,B 0,C 180,E1 -3033.903,E2 -3033.903} C_VEL
LIN {X 0,Y 559.148,Z 514.829,A -85,B 0,C 180,E1 -3036.567,E2 -3036.567} C_VEL
LIN {X 0,Y 559.177,Z 514.835,A -85,B 0,C 180,E1 -3039.395,E2 -3039.395} C_VEL
LIN {X 0,Y 559.147,Z 514.835,A -85,B 0,C 180,E1 -3041.686,E2 -3041.686} C_VEL
LIN {X 0,Y 559.161,Z 514.83,A -85,B 0,C 180,E1 -3043.948,E2 -3043.948} C_VEL
LIN {X 0,Y 559.163,Z 514.828,A -85,B 0,C 180,E1 -3046.184,E2 -3046.184} C_VEL
LIN {X 0,Y 559.201,Z 514.828,A -85,B 0,C 180,E1 -3049.134,E2 -3049.134} C_VEL
LIN {X 0,Y 559.201,Z 514.824,A -85,B 0,C 180,E1 -3052.054,E2 -3052.054} C_VEL
LIN {X 0,Y 559.251,Z 514.819,A -85,B 0,C 180,E1 -3054.953,E2 -3054.953} C_VEL
LIN {X 0,Y 559.243,Z 514.821,A -85,B 0,C 180,E1 -3057.839,E2 -3057.839} C_VEL
LIN {X 0,Y 559.267,Z 514.815,A -85,B 0,C 180,E1 -3060.72,E2 -3060.72} C_VEL
LIN {X 0,Y 559.237,Z 514.82,A -85,B 0,C 180,E1 -3062.881,E2 -3062.881} C_VEL
LIN {X 0,Y 559.221,Z 514.825,A -85,B 0,C 180,E1 -3065.77,E2 -3065.77} C_VEL
LIN {X 0,Y 559.194,Z 514.824,A -85,B 0,C 180,E1 -3068.674,E2 -3068.674} C_VEL
LIN {X 0,Y 559.2,Z 514.83,A -85,B 0,C 180,E1 -3071.601,E2 -3071.601} C_VEL
LIN {X 0,Y 559.189,Z 514.824,A -85,B 0,C 180,E1 -3074.596,E2 -3074.596} C_VEL
LIN {X 0,Y 559.155,Z 514.836,A -85,B 0,C 180,E1 -3077.557,E2 -3077.557} C_VEL
LIN {X 0,Y 559.166,Z 514.83,A -85,B 0,C 180,E1 -3079.838,E2 -3079.838} C_VEL
LIN {X 0,Y 559.135,Z 514.831,A -85,B 0,C 180,E1 -3082.153,E2 -3082.153} C_VEL
LIN {X 0,Y 559.172,Z 514.832,A -85,B 0,C 180,E1 -3085.188,E2 -3085.188} C_VEL
LIN {X 0,Y 559.188,Z 514.829,A -85,B 0,C 180,E1 -3087.712,E2 -3087.712} C_VEL
LIN {X 0,Y 559.146,Z 514.83,A -85,B 0,C 180,E1 -3090.631,E2 -3090.631} C_VEL
LIN {X 0,Y 558.483,Z 514.921,A -85,B 0,C 180,E1 -3091.232,E2 -3091.232} C_VEL
LIN {X 0,Y 555.621,Z 515.273,A -85,B 0,C 180,E1 -3092.208,E2 -3092.208} C_VEL
LIN {X 0,Y 553.21,Z 515.572,A -85,B 0,C 180,E1 -3092.994,E2 -3092.994} C_VEL
LIN {X 0,Y 552.191,Z 515.703,A -85,B 0,C 180,E1 -3093.601,E2 -3093.601} C_VEL
LIN {X 0,Y 552.118,Z 515.706,A -85,B 0,C 180,E1 -3093.806,E2 -3093.806} C_VEL
LIN {X 0,Y 552.107,Z 515.708,A -85,B 0,C 180,E1 -3096.747,E2 -3096.747} C_VEL
LIN {X 0,Y 552.145,Z 515.71,A -85,B 0,C 180,E1 -3099.526,E2 -3099.526} C_VEL
LIN {X 0,Y 552.126,Z 515.704,A -85,B 0,C 180,E1 -3102.426,E2 -3102.426} C_VEL
LIN {X 0,Y 552.097,Z 515.715,A -85,B 0,C 180,E1 -3105.564,E2 -3105.564} C_VEL
LIN {X 0,Y 552.139,Z 515.703,A -85,B 0,C 180,E1 -3108.677,E2 -3108.677} C_VEL
LIN {X 0,Y 552.119,Z 515.715,A -85,B 0,C 180,E1 -3111.412,E2 -3111.412} C_VEL
LIN {X 0,Y 552.101,Z 515.708,A -85,B 0,C 180,E1 -3114.158,E2 -3114.158} C_VEL
LIN {X 0,Y 552.121,Z 515.706,A -85,B 0,C 180,E1 -3116.815,E2 -3116.815} C_VEL
LIN {X 0,Y 552.106,Z 515.717,A -85,B 0,C 180,E1 -3119.392,E2 -3119.392} C_VEL
LIN {X 0,Y 552.121,Z 515.707,A -85,B 0,C 180,E1 -3121.903,E2 -3121.903} C_VEL
LIN {X 0,Y 552.158,Z 515.701,A -85,B 0,C 180,E1 -3124.65,E2 -3124.65} C_VEL
LIN {X 0,Y 552.095,Z 515.717,A -85,B 0,C 180,E1 -3127.55,E2 -3127.55} C_VEL
LIN {X 0,Y 552.152,Z 515.703,A -85,B 0,C 180,E1 -3130.374,E2 -3130.374} C_VEL
LIN {X 0,Y 552.16,Z 515.706,A -85,B 0,C 180,E1 -3132.978,E2 -3132.978} C_VEL
LIN {X 0,Y 552.198,Z 515.886,A -85,B 0,C 180,E1 -3133.977,E2 -3133.977} C_VEL
LIN {X 0,Y 552.628,Z 519.76,A -85,B 0,C 180,E1 -3134.718,E2 -3134.718} C_VEL
LIN {X 0,Y 552.339,Z 537.142,A -85,B 0,C 180,E1 -3137.881,E2 -3137.881} C_VEL
LIN {X 0,Y 552.191,Z 547.288,A -85,B 0,C 180,E1 -3139.69,E2 -3139.69} C_VEL
LIN {X 0,Y 553.396,Z 554.851,A -85,B 0,C 180,E1 -3139.821,E2 -3139.821} C_VEL
LIN {X 0,Y 553.129,Z 654.448,A -85,B 0,C 180,E1 -3141.138,E2 -3141.138} C_VEL
LIN {X 0,Y 552.991,Z 667.437,A -85,B 0,C 180,E1 -3141.458,E2 -3141.458} C_VEL
LIN {X 0,Y 552.814,Z 679.981,A -85,B 0,C 180,E1 -3141.915,E2 -3141.915} C_VEL
LIN {X 0,Y 552.666,Z 691.955,A -85,B 0,C 180,E1 -3142.511,E2 -3142.511} C_VEL
LIN {X 0,Y 552.444,Z 703.7,A -85,B 0,C 180,E1 -3143.266,E2 -3143.266} C_VEL
LIN {X 0,Y 552.295,Z 714.69,A -85,B 0,C 180,E1 -3144.157,E2 -3144.157} C_VEL
LIN {X 0,Y 552.189,Z 723.755,A -85,B 0,C 180,E1 -3145.072,E2 -3145.072} C_VEL
LIN {X 0,Y 551.982,Z 732.609,A -85,B 0,C 180,E1 -3146.167,E2 -3146.167} C_VEL
LIN {X 0,Y 551.856,Z 739.749,A -85,B 0,C 180,E1 -3147.263,E2 -3147.263} C_VEL
LIN {X 0,Y 551.795,Z 744.573,A -85,B 0,C 180,E1 -3148.175,E2 -3148.175} C_VEL
LIN {X 0,Y 551.673,Z 749.275,A -85,B 0,C 180,E1 -3149.27,E2 -3149.27} C_VEL
LIN {X 0,Y 551.731,Z 752.878,A -85,B 0,C 180,E1 -3150.365,E2 -3150.365} C_VEL
LIN {X 0,Y 551.646,Z 755.485,A -85,B 0,C 180,E1 -3151.46,E2 -3151.46} C_VEL
LIN {X 0,Y 551.656,Z 756.71,A -85,B 0,C 180,E1 -3152.19,E2 -3152.19} C_VEL
LIN {X 0,Y 551.718,Z 757.528,A -85,B 0,C 180,E1 -3152.921,E2 -3152.921} C_VEL
LIN {X 0,Y 551.731,Z 757.921,A -85,B 0,C 180,E1 -3153.652,E2 -3153.652} C_VEL
LIN {X 0,Y 551.68,Z 757.562,A -85,B 0,C 180,E1 -3155.116,E2 -3155.116} C_VEL
LIN {X 0,Y 551.73,Z 755.745,A -85,B 0,C 180,E1 -3156.496,E2 -3156.496} C_VEL
LIN {X 0,Y 551.731,Z 752.988,A -85,B 0,C 180,E1 -3157.686,E2 -3157.686} C_VEL
LIN {X 0,Y 551.763,Z 749.381,A -85,B 0,C 180,E1 -3158.792,E2 -3158.792} C_VEL
LIN {X 0,Y 551.824,Z 744.644,A -85,B 0,C 180,E1 -3159.9,E2 -3159.9} C_VEL
LIN {X 0,Y 551.927,Z 738.628,A -85,B 0,C 180,E1 -3161.011,E2 -3161.011} C_VEL
LIN {X 0,Y 551.991,Z 731.108,A -85,B 0,C 180,E1 -3162.127,E2 -3162.127} C_VEL
LIN {X 0,Y 552.127,Z 723.415,A -85,B 0,C 180,E1 -3163.058,E2 -3163.058} C_VEL
LIN {X 0,Y 552.294,Z 714.042,A -85,B 0,C 180,E1 -3163.991,E2 -3163.991} C_VEL
LIN {X 0,Y 552.423,Z 703.697,A -85,B 0,C 180,E1 -3164.825,E2 -3164.825} C_VEL
LIN {X 0,Y 552.654,Z 691.893,A -85,B 0,C 180,E1 -3165.583,E2 -3165.583} C_VEL
LIN {X 0,Y 552.856,Z 679.532,A -85,B 0,C 180,E1 -3166.193,E2 -3166.193} C_VEL
LIN {X 0,Y 552.987,Z 666.431,A -85,B 0,C 180,E1 -3166.663,E2 -3166.663} C_VEL
LIN {X 0,Y 553.113,Z 653.669,A -85,B 0,C 180,E1 -3166.968,E2 -3166.968} C_VEL
LIN {X 0,Y 553.256,Z 553.674,A -85,B 0,C 180,E1 -3168.288,E2 -3168.288} C_VEL
LIN {X 0,Y 552.255,Z 547.158,A -85,B 0,C 180,E1 -3168.406,E2 -3168.406} C_VEL
LIN {X 0,Y 552.453,Z 529.197,A -85,B 0,C 180,E1 -3171.649,E2 -3171.649} C_VEL
LIN {X 0,Y 552.542,Z 518.132,A -85,B 0,C 180,E1 -3173.68,E2 -3173.68} C_VEL
LIN {X 0,Y 552.161,Z 515.708,A -85,B 0,C 180,E1 -3174.185,E2 -3174.185} C_VEL
LIN {X 0,Y 552.141,Z 515.706,A -85,B 0,C 180,E1 -3177.272,E2 -3177.272} C_VEL
LIN {X 0,Y 552.119,Z 515.708,A -85,B 0,C 180,E1 -3180.05,E2 -3180.05} C_VEL
LIN {X 0,Y 552.127,Z 515.712,A -85,B 0,C 180,E1 -3182.848,E2 -3182.848} C_VEL
LIN {X 0,Y 552.094,Z 515.709,A -85,B 0,C 180,E1 -3185.442,E2 -3185.442} C_VEL
LIN {X 0,Y 552.097,Z 515.708,A -85,B 0,C 180,E1 -3187.885,E2 -3187.885} C_VEL
LIN {X 0,Y 552.14,Z 515.71,A -85,B 0,C 180,E1 -3190.477,E2 -3190.477} C_VEL
LIN {X 0,Y 552.114,Z 515.706,A -85,B 0,C 180,E1 -3193.483,E2 -3193.483} C_VEL
LIN {X 0,Y 552.116,Z 515.714,A -85,B 0,C 180,E1 -3196.577,E2 -3196.577} C_VEL
LIN {X 0,Y 552.118,Z 515.704,A -85,B 0,C 180,E1 -3199.519,E2 -3199.519} C_VEL
LIN {X 0,Y 552.088,Z 515.714,A -85,B 0,C 180,E1 -3202.335,E2 -3202.335} C_VEL
LIN {X 0,Y 552.126,Z 515.708,A -85,B 0,C 180,E1 -3205.054,E2 -3205.054} C_VEL
LIN {X 0,Y 552.122,Z 515.705,A -85,B 0,C 180,E1 -3207.681,E2 -3207.681} C_VEL
LIN {X 0,Y 552.139,Z 515.705,A -85,B 0,C 180,E1 -3210.236,E2 -3210.236} C_VEL
LIN {X 0,Y 552.14,Z 515.706,A -85,B 0,C 180,E1 -3212.997,E2 -3212.997} C_VEL
LIN {X 0,Y 552.105,Z 515.709,A -85,B 0,C 180,E1 -3215.161,E2 -3215.161} C_VEL
LIN {X 0,Y 552.089,Z 515.707,A -85,B 0,C 180,E1 -3217.549,E2 -3217.549} C_VEL
LIN {X 0,Y 552.14,Z 515.708,A -85,B 0,C 180,E1 -3220.373,E2 -3220.373} C_VEL
LIN {X 0,Y 552.149,Z 515.706,A -85,B 0,C 180,E1 -3222.977,E2 -3222.977} C_VEL
LIN {X 0,Y 552.127,Z 515.705,A -85,B 0,C 180,E1 -3226.004,E2 -3226.004} C_VEL
LIN {X 0,Y 552.169,Z 515.703,A -85,B 0,C 180,E1 -3228.993,E2 -3228.993} C_VEL
LIN {X 0,Y 552.157,Z 515.7,A -85,B 0,C 180,E1 -3231.951,E2 -3231.951} C_VEL
LIN {X 0,Y 552.225,Z 515.697,A -85,B 0,C 180,E1 -3234.889,E2 -3234.889} C_VEL
LIN {X 0,Y 552.215,Z 515.692,A -85,B 0,C 180,E1 -3237.812,E2 -3237.812} C_VEL
LIN {X 0,Y 552.237,Z 515.698,A -85,B 0,C 180,E1 -3240.729,E2 -3240.729} C_VEL
LIN {X 0,Y 552.203,Z 515.698,A -85,B 0,C 180,E1 -3242.918,E2 -3242.918} C_VEL
LIN {X 0,Y 552.191,Z 515.697,A -85,B 0,C 180,E1 -3245.844,E2 -3245.844} C_VEL
LIN {X 0,Y 552.162,Z 515.706,A -85,B 0,C 180,E1 -3248.786,E2 -3248.786} C_VEL
LIN {X 0,Y 552.155,Z 515.701,A -85,B 0,C 180,E1 -3251.751,E2 -3251.751} C_VEL
LIN {X 0,Y 552.126,Z 515.712,A -85,B 0,C 180,E1 -3254.749,E2 -3254.749} C_VEL
LIN {X 0,Y 552.106,Z 515.706,A -85,B 0,C 180,E1 -3257.789,E2 -3257.789} C_VEL
LIN {X 0,Y 552.125,Z 515.707,A -85,B 0,C 180,E1 -3260.101,E2 -3260.101} C_VEL
LIN {X 0,Y 552.088,Z 515.717,A -85,B 0,C 180,E1 -3262.451,E2 -3262.451} C_VEL
LIN {X 0,Y 552.148,Z 515.702,A -85,B 0,C 180,E1 -3265.351,E2 -3265.351} C_VEL
LIN {X 0,Y 552.119,Z 515.707,A -85,B 0,C 180,E1 -3268.098,E2 -3268.098} C_VEL
LIN {X 0,Y 552.106,Z 515.716,A -85,B 0,C 180,E1 -3270.609,E2 -3270.609} C_VEL
LIN {X 0,Y 552.122,Z 515.706,A -85,B 0,C 180,E1 -3273.185,E2 -3273.185} C_VEL
LIN {X 0,Y 552.107,Z 515.707,A -85,B 0,C 180,E1 -3275.842,E2 -3275.842} C_VEL
LIN {X 0,Y 552.12,Z 515.708,A -85,B 0,C 180,E1 -3279.063,E2 -3279.063} C_VEL
LIN {X 0,Y 552.134,Z 515.704,A -85,B 0,C 180,E1 -3281.445,E2 -3281.445} C_VEL
LIN {X 0,Y 552.091,Z 515.719,A -85,B 0,C 180,E1 -3284.533,E2 -3284.533} C_VEL
LIN {X 0,Y 552.127,Z 515.705,A -85,B 0,C 180,E1 -3287.585,E2 -3287.585} C_VEL
LIN {X 0,Y 552.147,Z 515.711,A -85,B 0,C 180,E1 -3290.475,E2 -3290.475} C_VEL
LIN {X 0,Y 552.108,Z 515.707,A -85,B 0,C 180,E1 -3293.317,E2 -3293.317} C_VEL
LIN {X 0,Y 552.126,Z 515.706,A -85,B 0,C 180,E1 -3295.94,E2 -3295.94} C_VEL
LIN {X 0,Y 552.118,Z 515.715,A -85,B 0,C 180,E1 -3298.541,E2 -3298.541} C_VEL
LIN {X 0,Y 552.124,Z 515.706,A -85,B 0,C 180,E1 -3301.439,E2 -3301.439} C_VEL
LIN {X 0,Y 552.13,Z 515.713,A -85,B 0,C 180,E1 -3304.356,E2 -3304.356} C_VEL
LIN {X 0,Y 552.146,Z 515.884,A -85,B 0,C 180,E1 -3306.464,E2 -3306.464} C_VEL
LIN {X 0,Y 553.214,Z 521.633,A -85,B 0,C 180,E1 -3307.401,E2 -3307.401} C_VEL
LIN {X 0,Y 552.887,Z 541.425,A -85,B 0,C 180,E1 -3310.428,E2 -3310.428} C_VEL
LIN {X 0,Y 552.591,Z 558.322,A -85,B 0,C 180,E1 -3312.992,E2 -3312.992} C_VEL
LIN {X 0,Y 552.366,Z 575.89,A -85,B 0,C 180,E1 -3315.626,E2 -3315.626} C_VEL
LIN {X 0,Y 553.44,Z 583.803,A -85,B 0,C 180,E1 -3315.763,E2 -3315.763} C_VEL
LIN {X 0,Y 553.117,Z 683.962,A -85,B 0,C 180,E1 -3317.083,E2 -3317.083} C_VEL
LIN {X 0,Y 552.985,Z 697.228,A -85,B 0,C 180,E1 -3317.406,E2 -3317.406} C_VEL
LIN {X 0,Y 552.849,Z 710.494,A -85,B 0,C 180,E1 -3317.892,E2 -3317.892} C_VEL
LIN {X 0,Y 552.677,Z 722.745,A -85,B 0,C 180,E1 -3318.512,E2 -3318.512} C_VEL
LIN {X 0,Y 552.464,Z 734.488,A -85,B 0,C 180,E1 -3319.278,E2 -3319.278} C_VEL
LIN {X 0,Y 552.276,Z 744.649,A -85,B 0,C 180,E1 -3320.108,E2 -3320.108} C_VEL
LIN {X 0,Y 552.103,Z 753.788,A -85,B 0,C 180,E1 -3321.029,E2 -3321.029} C_VEL
LIN {X 0,Y 551.96,Z 762.69,A -85,B 0,C 180,E1 -3322.133,E2 -3322.133} C_VEL
LIN {X 0,Y 551.835,Z 769.85,A -85,B 0,C 180,E1 -3323.235,E2 -3323.235} C_VEL
LIN {X 0,Y 551.804,Z 776.366,A -85,B 0,C 180,E1 -3324.519,E2 -3324.519} C_VEL
LIN {X 0,Y 551.764,Z 780.677,A -85,B 0,C 180,E1 -3325.617,E2 -3325.617} C_VEL
LIN {X 0,Y 551.75,Z 782.958,A -85,B 0,C 180,E1 -3326.349,E2 -3326.349} C_VEL
LIN {X 0,Y 551.724,Z 784.808,A -85,B 0,C 180,E1 -3327.079,E2 -3327.079} C_VEL
LIN {X 0,Y 551.645,Z 787.184,A -85,B 0,C 180,E1 -3328.54,E2 -3328.54} C_VEL
LIN {X 0,Y 551.64,Z 788,A -85,B 0,C 180,E1 -3330,E2 -3330} C_VEL
LIN {X 0,Y 551.645,Z 787.185,A -85,B 0,C 180,E1 -3331.46,E2 -3331.46} C_VEL
LIN {X 0,Y 551.724,Z 784.81,A -85,B 0,C 180,E1 -3332.921,E2 -3332.921} C_VEL
LIN {X 0,Y 551.763,Z 781.896,A -85,B 0,C 180,E1 -3334.017,E2 -3334.017} C_VEL
LIN {X 0,Y 551.724,Z 777.949,A -85,B 0,C 180,E1 -3335.116,E2 -3335.116} C_VEL
LIN {X 0,Y 551.803,Z 772.189,A -85,B 0,C 180,E1 -3336.341,E2 -3336.341} C_VEL
LIN {X 0,Y 551.926,Z 765.238,A -85,B 0,C 180,E1 -3337.499,E2 -3337.499} C_VEL
LIN {X 0,Y 552.082,Z 756.993,A -85,B 0,C 180,E1 -3338.602,E2 -3338.602} C_VEL
LIN {X 0,Y 552.222,Z 748.541,A -85,B 0,C 180,E1 -3339.523,E2 -3339.523} C_VEL
LIN {X 0,Y 552.412,Z 738.098,A -85,B 0,C 180,E1 -3340.445,E2 -3340.445} C_VEL
LIN {X 0,Y 552.602,Z 727.134,A -85,B 0,C 180,E1 -3341.224,E2 -3341.224} C_VEL
LIN {X 0,Y 552.752,Z 716.413,A -85,B 0,C 180,E1 -3341.831,E2 -3341.831} C_VEL
LIN {X 0,Y 552.902,Z 704.772,A -85,B 0,C 180,E1 -3342.339,E2 -3342.339} C_VEL
LIN {X 0,Y 553.017,Z 691.358,A -85,B 0,C 180,E1 -3342.756,E2 -3342.756} C_VEL
LIN {X 0,Y 553.173,Z 678.106,A -85,B 0,C 180,E1 -3343.009,E2 -3343.009} C_VEL
LIN {X 0,Y 553.32,Z 582.023,A -85,B 0,C 180,E1 -3344.263,E2 -3344.263} C_VEL
LIN {X 0,Y 552.378,Z 575.774,A -85,B 0,C 180,E1 -3344.391,E2 -3344.391} C_VEL
LIN {X 0,Y 552.665,Z 555.098,A -85,B 0,C 180,E1 -3347.494,E2 -3347.494} C_VEL
LIN {X 0,Y 553.019,Z 534.366,A -85,B 0,C 180,E1 -3350.649,E2 -3350.649} C_VEL
LIN {X 0,Y 553.214,Z 521.637,A -85,B 0,C 180,E1 -3352.599,E2 -3352.599} C_VEL
LIN {X 0,Y 552.123,Z 515.714,A -85,B 0,C 180,E1 -3353.581,E2 -3353.581} C_VEL
LIN {X 0,Y 552.12,Z 515.707,A -85,B 0,C 180,E1 -3356.456,E2 -3356.456} C_VEL
LIN {X 0,Y 552.11,Z 515.709,A -85,B 0,C 180,E1 -3358.928,E2 -3358.928} C_VEL
LIN {X 0,Y 552.135,Z 515.713,A -85,B 0,C 180,E1 -3361.479,E2 -3361.479} C_VEL
LIN {X 0,Y 552.133,Z 515.704,A -85,B 0,C 180,E1 -3364.17,E2 -3364.17} C_VEL
LIN {X 0,Y 552.106,Z 515.707,A -85,B 0,C 180,E1 -3366.746,E2 -3366.746} C_VEL
LIN {X 0,Y 552.147,Z 515.711,A -85,B 0,C 180,E1 -3369.525,E2 -3369.525} C_VEL
LIN {X 0,Y 552.127,Z 515.704,A -85,B 0,C 180,E1 -3372.424,E2 -3372.424} C_VEL
LIN {X 0,Y 552.093,Z 515.716,A -85,B 0,C 180,E1 -3375.562,E2 -3375.562} C_VEL
LIN {X 0,Y 552.135,Z 515.703,A -85,B 0,C 180,E1 -3378.675,E2 -3378.675} C_VEL
LIN {X 0,Y 552.114,Z 515.715,A -85,B 0,C 180,E1 -3381.411,E2 -3381.411} C_VEL
LIN {X 0,Y 552.107,Z 515.707,A -85,B 0,C 180,E1 -3384.158,E2 -3384.158} C_VEL
LIN {X 0,Y 552.122,Z 515.706,A -85,B 0,C 180,E1 -3386.815,E2 -3386.815} C_VEL
LIN {X 0,Y 552.106,Z 515.715,A -85,B 0,C 180,E1 -3389.391,E2 -3389.391} C_VEL
LIN {X 0,Y 552.119,Z 515.708,A -85,B 0,C 180,E1 -3391.902,E2 -3391.902} C_VEL
LIN {X 0,Y 552.148,Z 515.701,A -85,B 0,C 180,E1 -3394.649,E2 -3394.649} C_VEL
LIN {X 0,Y 552.088,Z 515.717,A -85,B 0,C 180,E1 -3397.549,E2 -3397.549} C_VEL
LIN {X 0,Y 552.14,Z 515.702,A -85,B 0,C 180,E1 -3400.373,E2 -3400.373} C_VEL
LIN {X 0,Y 552.148,Z 515.704,A -85,B 0,C 180,E1 -3402.977,E2 -3402.977} C_VEL
LIN {X 0,Y 552.126,Z 515.706,A -85,B 0,C 180,E1 -3406.004,E2 -3406.004} C_VEL
LIN {X 0,Y 552.168,Z 515.702,A -85,B 0,C 180,E1 -3408.994,E2 -3408.994} C_VEL
LIN {X 0,Y 552.155,Z 515.703,A -85,B 0,C 180,E1 -3411.952,E2 -3411.952} C_VEL
LIN {X 0,Y 552.225,Z 515.694,A -85,B 0,C 180,E1 -3414.889,E2 -3414.889} C_VEL
LIN {X 0,Y 552.214,Z 515.697,A -85,B 0,C 180,E1 -3417.812,E2 -3417.812} C_VEL
LIN {X 0,Y 552.237,Z 515.691,A -85,B 0,C 180,E1 -3420.729,E2 -3420.729} C_VEL
LIN {X 0,Y 552.202,Z 515.697,A -85,B 0,C 180,E1 -3422.918,E2 -3422.918} C_VEL
LIN {X 0,Y 552.191,Z 515.699,A -85,B 0,C 180,E1 -3425.844,E2 -3425.844} C_VEL
LIN {X 0,Y 552.162,Z 515.701,A -85,B 0,C 180,E1 -3428.786,E2 -3428.786} C_VEL
LIN {X 0,Y 552.155,Z 515.705,A -85,B 0,C 180,E1 -3431.751,E2 -3431.751} C_VEL
LIN {X 0,Y 552.127,Z 515.705,A -85,B 0,C 180,E1 -3434.749,E2 -3434.749} C_VEL
LIN {X 0,Y 552.106,Z 515.711,A -85,B 0,C 180,E1 -3437.789,E2 -3437.789} C_VEL
LIN {X 0,Y 552.126,Z 515.705,A -85,B 0,C 180,E1 -3440.102,E2 -3440.102} C_VEL
LIN {X 0,Y 552.089,Z 515.709,A -85,B 0,C 180,E1 -3442.451,E2 -3442.451} C_VEL
LIN {X 0,Y 552.149,Z 515.71,A -85,B 0,C 180,E1 -3445.352,E2 -3445.352} C_VEL
LIN {X 0,Y 552.12,Z 515.706,A -85,B 0,C 180,E1 -3448.098,E2 -3448.098} C_VEL
LIN {X 0,Y 552.106,Z 515.707,A -85,B 0,C 180,E1 -3450.626,E2 -3450.626} C_VEL
LIN {X 0,Y 552.123,Z 515.71,A -85,B 0,C 180,E1 -3453.186,E2 -3453.186} C_VEL
LIN {X 0,Y 552.118,Z 515.706,A -85,B 0,C 180,E1 -3453.806,E2 -3453.806} C_VEL
LIN {X 0,Y 551.483,Z 515.788,A -85,B 0,C 180,E1 -3454.415,E2 -3454.415} C_VEL
LIN {X 0,Y 548.657,Z 516.146,A -85,B 0,C 180,E1 -3455.403,E2 -3455.403} C_VEL
LIN {X 0,Y 546.232,Z 516.442,A -85,B 0,C 180,E1 -3456.198,E2 -3456.198} C_VEL
LIN {X 0,Y 545.161,Z 516.574,A -85,B 0,C 180,E1 -3456.812,E2 -3456.812} C_VEL
LIN {X 0,Y 545.059,Z 516.588,A -85,B 0,C 180,E1 -3457.02,E2 -3457.02} C_VEL
LIN {X 0,Y 545.072,Z 516.583,A -85,B 0,C 180,E1 -3460.142,E2 -3460.142} C_VEL
LIN {X 0,Y 545.08,Z 516.587,A -85,B 0,C 180,E1 -3463.107,E2 -3463.107} C_VEL
LIN {X 0,Y 545.063,Z 516.584,A -85,B 0,C 180,E1 -3466.225,E2 -3466.225} C_VEL
LIN {X 0,Y 545.1,Z 516.582,A -85,B 0,C 180,E1 -3468.888,E2 -3468.888} C_VEL
LIN {X 0,Y 545.053,Z 516.589,A -85,B 0,C 180,E1 -3471.764,E2 -3471.764} C_VEL
LIN {X 0,Y 545.051,Z 516.585,A -85,B 0,C 180,E1 -3474.534,E2 -3474.534} C_VEL
LIN {X 0,Y 545.08,Z 516.589,A -85,B 0,C 180,E1 -3477.213,E2 -3477.213} C_VEL
LIN {X 0,Y 545.066,Z 516.587,A -85,B 0,C 180,E1 -3479.811,E2 -3479.811} C_VEL
LIN {X 0,Y 545.091,Z 516.58,A -85,B 0,C 180,E1 -3482.345,E2 -3482.345} C_VEL
LIN {X 0,Y 545.119,Z 516.579,A -85,B 0,C 180,E1 -3484.821,E2 -3484.821} C_VEL
LIN {X 0,Y 545.039,Z 516.594,A -85,B 0,C 180,E1 -3487.243,E2 -3487.243} C_VEL
LIN {X 0,Y 545.124,Z 516.579,A -85,B 0,C 180,E1 -3490.416,E2 -3490.416} C_VEL
LIN {X 0,Y 545.113,Z 516.587,A -85,B 0,C 180,E1 -3493.763,E2 -3493.763} C_VEL
LIN {X 0,Y 545.601,Z 519.092,A -85,B 0,C 180,E1 -3494.306,E2 -3494.306} C_VEL
LIN {X 0,Y 545.394,Z 534.353,A -85,B 0,C 180,E1 -3497.157,E2 -3497.157} C_VEL
LIN {X 0,Y 545.19,Z 547.115,A -85,B 0,C 180,E1 -3499.486,E2 -3499.486} C_VEL
LIN {X 0,Y 546.536,Z 555.874,A -85,B 0,C 180,E1 -3499.652,E2 -3499.652} C_VEL
LIN {X 0,Y 546.243,Z 653.611,A -85,B 0,C 180,E1 -3500.955,E2 -3500.955} C_VEL
LIN {X 0,Y 546.081,Z 666.891,A -85,B 0,C 180,E1 -3501.279,E2 -3501.279} C_VEL
LIN {X 0,Y 545.874,Z 680.137,A -85,B 0,C 180,E1 -3501.765,E2 -3501.765} C_VEL
LIN {X 0,Y 545.715,Z 691.279,A -85,B 0,C 180,E1 -3502.322,E2 -3502.322} C_VEL
LIN {X 0,Y 545.462,Z 703.436,A -85,B 0,C 180,E1 -3503.107,E2 -3503.107} C_VEL
LIN {X 0,Y 545.299,Z 714.258,A -85,B 0,C 180,E1 -3503.989,E2 -3503.989} C_VEL
LIN {X 0,Y 545.16,Z 722.592,A -85,B 0,C 180,E1 -3504.823,E2 -3504.823} C_VEL
LIN {X 0,Y 544.914,Z 731.65,A -85,B 0,C 180,E1 -3505.932,E2 -3505.932} C_VEL
LIN {X 0,Y 544.752,Z 738.96,A -85,B 0,C 180,E1 -3507.042,E2 -3507.042} C_VEL
LIN {X 0,Y 544.713,Z 744.83,A -85,B 0,C 180,E1 -3508.152,E2 -3508.152} C_VEL
LIN {X 0,Y 544.577,Z 749.477,A -85,B 0,C 180,E1 -3509.261,E2 -3509.261} C_VEL
LIN {X 0,Y 544.639,Z 753.029,A -85,B 0,C 180,E1 -3510.37,E2 -3510.37} C_VEL
LIN {X 0,Y 544.547,Z 755.588,A -85,B 0,C 180,E1 -3511.479,E2 -3511.479} C_VEL
LIN {X 0,Y 544.57,Z 756.789,A -85,B 0,C 180,E1 -3512.219,E2 -3512.219} C_VEL
LIN {X 0,Y 544.645,Z 757.562,A -85,B 0,C 180,E1 -3512.959,E2 -3512.959} C_VEL
LIN {X 0,Y 544.645,Z 757.932,A -85,B 0,C 180,E1 -3513.699,E2 -3513.699} C_VEL
LIN {X 0,Y 544.599,Z 757.527,A -85,B 0,C 180,E1 -3515.183,E2 -3515.183} C_VEL
LIN {X 0,Y 544.635,Z 755.845,A -85,B 0,C 180,E1 -3516.477,E2 -3516.477} C_VEL
LIN {X 0,Y 544.649,Z 752.836,A -85,B 0,C 180,E1 -3517.787,E2 -3517.787} C_VEL
LIN {X 0,Y 544.676,Z 749.177,A -85,B 0,C 180,E1 -3518.907,E2 -3518.907} C_VEL
LIN {X 0,Y 544.734,Z 744.382,A -85,B 0,C 180,E1 -3520.03,E2 -3520.03} C_VEL
LIN {X 0,Y 544.845,Z 738.305,A -85,B 0,C 180,E1 -3521.156,E2 -3521.156} C_VEL
LIN {X 0,Y 544.94,Z 730.715,A -85,B 0,C 180,E1 -3522.286,E2 -3522.286} C_VEL
LIN {X 0,Y 545.117,Z 722.945,A -85,B 0,C 180,E1 -3523.229,E2 -3523.229} C_VEL
LIN {X 0,Y 545.29,Z 713.429,A -85,B 0,C 180,E1 -3524.175,E2 -3524.175} C_VEL
LIN {X 0,Y 545.451,Z 702.814,A -85,B 0,C 180,E1 -3525.028,E2 -3525.028} C_VEL
LIN {X 0,Y 545.705,Z 690.96,A -85,B 0,C 180,E1 -3525.787,E2 -3525.787} C_VEL
LIN {X 0,Y 545.9,Z 679.369,A -85,B 0,C 180,E1 -3526.357,E2 -3526.357} C_VEL
LIN {X 0,Y 546.049,Z 666.21,A -85,B 0,C 180,E1 -3526.833,E2 -3526.833} C_VEL
LIN {X 0,Y 546.217,Z 653.314,A -85,B 0,C 180,E1 -3527.141,E2 -3527.141} C_VEL
LIN {X 0,Y 546.46,Z 555.002,A -85,B 0,C 180,E1 -3528.451,E2 -3528.451} C_VEL
LIN {X 0,Y 545.176,Z 547.111,A -85,B 0,C 180,E1 -3528.606,E2 -3528.606} C_VEL
LIN {X 0,Y 545.438,Z 531.099,A -85,B 0,C 180,E1 -3531.537,E2 -3531.537} C_VEL
LIN {X 0,Y 545.634,Z 520.44,A -85,B 0,C 180,E1 -3533.533,E2 -3533.533} C_VEL
LIN {X 0,Y 545.114,Z 516.587,A -85,B 0,C 180,E1 -3534.288,E2 -3534.288} C_VEL
LIN {X 0,Y 545.095,Z 516.585,A -85,B 0,C 180,E1 -3537.173,E2 -3537.173} C_VEL
LIN {X 0,Y 545.066,Z 516.586,A -85,B 0,C 180,E1 -3539.338,E2 -3539.338} C_VEL
LIN {X 0,Y 545.06,Z 516.586,A -85,B 0,C 180,E1 -3541.914,E2 -3541.914} C_VEL
LIN {X 0,Y 545.077,Z 516.591,A -85,B 0,C 180,E1 -3544.562,E2 -3544.562} C_VEL
LIN {X 0,Y 545.038,Z 516.589,A -85,B 0,C 180,E1 -3547.303,E2 -3547.303} C_VEL
LIN {X 0,Y 545.091,Z 516.583,A -85,B 0,C 180,E1 -3550.139,E2 -3550.139} C_VEL
LIN {X 0,Y 545.085,Z 516.585,A -85,B 0,C 180,E1 -3553.105,E2 -3553.105} C_VEL
LIN {X 0,Y 545.061,Z 516.587,A -85,B 0,C 180,E1 -3556.224,E2 -3556.224} C_VEL
LIN {X 0,Y 545.093,Z 516.585,A -85,B 0,C 180,E1 -3558.886,E2 -3558.886} C_VEL
LIN {X 0,Y 545.048,Z 516.586,A -85,B 0,C 180,E1 -3561.762,E2 -3561.762} C_VEL
LIN {X 0,Y 545.061,Z 516.592,A -85,B 0,C 180,E1 -3564.533,E2 -3564.533} C_VEL
LIN {X 0,Y 545.077,Z 516.585,A -85,B 0,C 180,E1 -3567.212,E2 -3567.212} C_VEL
LIN {X 0,Y 545.095,Z 516.579,A -85,B 0,C 180,E1 -3569.812,E2 -3569.812} C_VEL
LIN {X 0,Y 545.094,Z 516.586,A -85,B 0,C 180,E1 -3572.824,E2 -3572.824} C_VEL
LIN {X 0,Y 545.044,Z 516.587,A -85,B 0,C 180,E1 -3575.63,E2 -3575.63} C_VEL
LIN {X 0,Y 545.062,Z 516.591,A -85,B 0,C 180,E1 -3578.836,E2 -3578.836} C_VEL
LIN {X 0,Y 545.076,Z 516.583,A -85,B 0,C 180,E1 -3581.195,E2 -3581.195} C_VEL
LIN {X 0,Y 545.068,Z 516.583,A -85,B 0,C 180,E1 -3583.521,E2 -3583.521} C_VEL
LIN {X 0,Y 545.086,Z 516.581,A -85,B 0,C 180,E1 -3585.82,E2 -3585.82} C_VEL
LIN {X 0,Y 545.123,Z 516.583,A -85,B 0,C 180,E1 -3588.849,E2 -3588.849} C_VEL
LIN {X 0,Y 545.127,Z 516.576,A -85,B 0,C 180,E1 -3591.847,E2 -3591.847} C_VEL
LIN {X 0,Y 545.2,Z 516.574,A -85,B 0,C 180,E1 -3594.823,E2 -3594.823} C_VEL
LIN {X 0,Y 545.186,Z 516.567,A -85,B 0,C 180,E1 -3597.784,E2 -3597.784} C_VEL
LIN {X 0,Y 545.207,Z 516.574,A -85,B 0,C 180,E1 -3600.739,E2 -3600.739} C_VEL
LIN {X 0,Y 545.169,Z 516.573,A -85,B 0,C 180,E1 -3602.956,E2 -3602.956} C_VEL
LIN {X 0,Y 545.163,Z 516.573,A -85,B 0,C 180,E1 -3605.92,E2 -3605.92} C_VEL
LIN {X 0,Y 545.119,Z 516.581,A -85,B 0,C 180,E1 -3608.9,E2 -3608.9} C_VEL
LIN {X 0,Y 545.126,Z 516.577,A -85,B 0,C 180,E1 -3611.904,E2 -3611.904} C_VEL
LIN {X 0,Y 545.076,Z 516.587,A -85,B 0,C 180,E1 -3614.944,E2 -3614.944} C_VEL
LIN {X 0,Y 545.074,Z 516.584,A -85,B 0,C 180,E1 -3618.026,E2 -3618.026} C_VEL
LIN {X 0,Y 545.09,Z 516.587,A -85,B 0,C 180,E1 -3620.372,E2 -3620.372} C_VEL
LIN {X 0,Y 545.082,Z 516.581,A -85,B 0,C 180,E1 -3623.559,E2 -3623.559} C_VEL
LIN {X 0,Y 545.081,Z 516.584,A -85,B 0,C 180,E1 -3626.001,E2 -3626.001} C_VEL
LIN {X 0,Y 545.085,Z 516.588,A -85,B 0,C 180,E1 -3628.75,E2 -3628.75} C_VEL
LIN {X 0,Y 545.07,Z 516.583,A -85,B 0,C 180,E1 -3631.683,E2 -3631.683} C_VEL
LIN {X 0,Y 545.079,Z 516.592,A -85,B 0,C 180,E1 -3634.563,E2 -3634.563} C_VEL
LIN {X 0,Y 545.033,Z 516.589,A -85,B 0,C 180,E1 -3637.304,E2 -3637.304} C_VEL
LIN {X 0,Y 545.087,Z 516.585,A -85,B 0,C 180,E1 -3640.141,E2 -3640.141} C_VEL
LIN {X 0,Y 545.073,Z 516.585,A -85,B 0,C 180,E1 -3643.107,E2 -3643.107} C_VEL
LIN {X 0,Y 545.061,Z 516.589,A -85,B 0,C 180,E1 -3646.225,E2 -3646.225} C_VEL
LIN {X 0,Y 545.094,Z 516.585,A -85,B 0,C 180,E1 -3648.888,E2 -3648.888} C_VEL
LIN {X 0,Y 545.086,Z 516.587,A -85,B 0,C 180,E1 -3650.82,E2 -3650.82} C_VEL
LIN {X 0,Y 545.046,Z 516.587,A -85,B 0,C 180,E1 -3653.621,E2 -3653.621} C_VEL
LIN {X 0,Y 545.068,Z 516.591,A -85,B 0,C 180,E1 -3656.329,E2 -3656.329} C_VEL
LIN {X 0,Y 545.067,Z 516.588,A -85,B 0,C 180,E1 -3658.953,E2 -3658.953} C_VEL
LIN {X 0,Y 545.102,Z 516.581,A -85,B 0,C 180,E1 -3661.508,E2 -3661.508} C_VEL
LIN {X 0,Y 545.095,Z 516.59,A -85,B 0,C 180,E1 -3664.492,E2 -3664.492} C_VEL
LIN {X 0,Y 545.103,Z 516.781,A -85,B 0,C 180,E1 -3666.309,E2 -3666.309} C_VEL
LIN {X 0,Y 546.291,Z 523.865,A -85,B 0,C 180,E1 -3667.472,E2 -3667.472} C_VEL
LIN {X 0,Y 545.893,Z 543.108,A -85,B 0,C 180,E1 -3670.444,E2 -3670.444} C_VEL
LIN {X 0,Y 545.6,Z 559.581,A -85,B 0,C 180,E1 -3672.96,E2 -3672.96} C_VEL
LIN {X 0,Y 545.394,Z 576.151,A -85,B 0,C 180,E1 -3675.447,E2 -3675.447} C_VEL
LIN {X 0,Y 546.574,Z 584.663,A -85,B 0,C 180,E1 -3675.592,E2 -3675.592} C_VEL
LIN {X 0,Y 546.208,Z 683.962,A -85,B 0,C 180,E1 -3676.916,E2 -3676.916} C_VEL
LIN {X 0,Y 546.07,Z 697.227,A -85,B 0,C 180,E1 -3677.244,E2 -3677.244} C_VEL
LIN {X 0,Y 545.894,Z 710.495,A -85,B 0,C 180,E1 -3677.736,E2 -3677.736} C_VEL
LIN {X 0,Y 545.727,Z 722.37,A -85,B 0,C 180,E1 -3678.342,E2 -3678.342} C_VEL
LIN {X 0,Y 545.478,Z 734.489,A -85,B 0,C 180,E1 -3679.139,E2 -3679.139} C_VEL
LIN {X 0,Y 545.257,Z 744.649,A -85,B 0,C 180,E1 -3679.979,E2 -3679.979} C_VEL
LIN {X 0,Y 545.078,Z 753.788,A -85,B 0,C 180,E1 -3680.913,E2 -3680.913} C_VEL
LIN {X 0,Y 544.916,Z 762.69,A -85,B 0,C 180,E1 -3682.031,E2 -3682.031} C_VEL
LIN {X 0,Y 544.784,Z 769.85,A -85,B 0,C 180,E1 -3683.147,E2 -3683.147} C_VEL
LIN {X 0,Y 544.741,Z 776.366,A -85,B 0,C 180,E1 -3684.447,E2 -3684.447} C_VEL
LIN {X 0,Y 544.66,Z 780.677,A -85,B 0,C 180,E1 -3685.56,E2 -3685.56} C_VEL
LIN {X 0,Y 544.669,Z 782.958,A -85,B 0,C 180,E1 -3686.301,E2 -3686.301} C_VEL
LIN {X 0,Y 544.65,Z 784.808,A -85,B 0,C 180,E1 -3687.041,E2 -3687.041} C_VEL
LIN {X 0,Y 544.546,Z 787.184,A -85,B 0,C 180,E1 -3688.521,E2 -3688.521} C_VEL
LIN {X 0,Y 544.541,Z 788,A -85,B 0,C 180,E1 -3690,E2 -3690} C_VEL
LIN {X 0,Y 544.546,Z 787.185,A -85,B 0,C 180,E1 -3691.479,E2 -3691.479} C_VEL
LIN {X 0,Y 544.65,Z 784.81,A -85,B 0,C 180,E1 -3692.959,E2 -3692.959} C_VEL
LIN {X 0,Y 544.683,Z 781.896,A -85,B 0,C 180,E1 -3694.069,E2 -3694.069} C_VEL
LIN {X 0,Y 544.654,Z 777.949,A -85,B 0,C 180,E1 -3695.182,E2 -3695.182} C_VEL
LIN {X 0,Y 544.739,Z 772.704,A -85,B 0,C 180,E1 -3696.328,E2 -3696.328} C_VEL
LIN {X 0,Y 544.836,Z 766.468,A -85,B 0,C 180,E1 -3697.411,E2 -3697.411} C_VEL
LIN {X 0,Y 545.006,Z 758.479,A -85,B 0,C 180,E1 -3698.528,E2 -3698.528} C_VEL
LIN {X 0,Y 545.152,Z 750.336,A -85,B 0,C 180,E1 -3699.46,E2 -3699.46} C_VEL
LIN {X 0,Y 545.362,Z 740.401,A -85,B 0,C 180,E1 -3700.394,E2 -3700.394} C_VEL
LIN {X 0,Y 545.571,Z 729.543,A -85,B 0,C 180,E1 -3701.211,E2 -3701.211} C_VEL
LIN {X 0,Y 545.763,Z 718.178,A -85,B 0,C 180,E1 -3701.89,E2 -3701.89} C_VEL
LIN {X 0,Y 545.937,Z 705.982,A -85,B 0,C 180,E1 -3702.452,E2 -3702.452} C_VEL
LIN {X 0,Y 546.09,Z 693.186,A -85,B 0,C 180,E1 -3702.874,E2 -3702.874} C_VEL
LIN {X 0,Y 546.27,Z 679.621,A -85,B 0,C 180,E1 -3703.153,E2 -3703.153} C_VEL
LIN {X 0,Y 546.447,Z 582.587,A -85,B 0,C 180,E1 -3704.439,E2 -3704.439} C_VEL
LIN {X 0,Y 545.372,Z 575.776,A -85,B 0,C 180,E1 -3704.58,E2 -3704.58} C_VEL
LIN {X 0,Y 545.694,Z 554.934,A -85,B 0,C 180,E1 -3707.75,E2 -3707.75} C_VEL
LIN {X 0,Y 546.058,Z 535.474,A -85,B 0,C 180,E1 -3710.728,E2 -3710.728} C_VEL
LIN {X 0,Y 546.251,Z 522.737,A -85,B 0,C 180,E1 -3712.704,E2 -3712.704} C_VEL
LIN {X 0,Y 545.08,Z 516.591,A -85,B 0,C 180,E1 -3713.731,E2 -3713.731} C_VEL
LIN {X 0,Y 545.08,Z 516.586,A -85,B 0,C 180,E1 -3716,E2 -3716} C_VEL
LIN {X 0,Y 545.089,Z 516.583,A -85,B 0,C 180,E1 -3718.748,E2 -3718.748} C_VEL
LIN {X 0,Y 545.077,Z 516.588,A -85,B 0,C 180,E1 -3721.682,E2 -3721.682} C_VEL
LIN {X 0,Y 545.074,Z 516.582,A -85,B 0,C 180,E1 -3724.563,E2 -3724.563} C_VEL
LIN {X 0,Y 545.036,Z 516.594,A -85,B 0,C 180,E1 -3727.303,E2 -3727.303} C_VEL
LIN {X 0,Y 545.073,Z 516.584,A -85,B 0,C 180,E1 -3730.141,E2 -3730.141} C_VEL
LIN {X 0,Y 545.083,Z 516.586,A -85,B 0,C 180,E1 -3733.105,E2 -3733.105} C_VEL
LIN {X 0,Y 545.062,Z 516.584,A -85,B 0,C 180,E1 -3736.223,E2 -3736.223} C_VEL
LIN {X 0,Y 545.096,Z 516.582,A -85,B 0,C 180,E1 -3738.887,E2 -3738.887} C_VEL
LIN {X 0,Y 545.048,Z 516.591,A -85,B 0,C 180,E1 -3741.762,E2 -3741.762} C_VEL
LIN {X 0,Y 545.059,Z 516.584,A -85,B 0,C 180,E1 -3744.533,E2 -3744.533} C_VEL
LIN {X 0,Y 545.076,Z 516.588,A -85,B 0,C 180,E1 -3747.212,E2 -3747.212} C_VEL
LIN {X 0,Y 545.094,Z 516.584,A -85,B 0,C 180,E1 -3749.812,E2 -3749.812} C_VEL
LIN {X 0,Y 545.093,Z 516.581,A -85,B 0,C 180,E1 -3752.824,E2 -3752.824} C_VEL
LIN {X 0,Y 545.044,Z 516.593,A -85,B 0,C 180,E1 -3755.63,E2 -3755.63} C_VEL
LIN {X 0,Y 545.06,Z 516.586,A -85,B 0,C 180,E1 -3758.836,E2 -3758.836} C_VEL
LIN {X 0,Y 545.076,Z 516.588,A -85,B 0,C 180,E1 -3761.195,E2 -3761.195} C_VEL
LIN {X 0,Y 545.068,Z 516.592,A -85,B 0,C 180,E1 -3763.521,E2 -3763.521} C_VEL
LIN {X 0,Y 545.085,Z 516.585,A -85,B 0,C 180,E1 -3765.82,E2 -3765.82} C_VEL
LIN {X 0,Y 545.122,Z 516.578,A -85,B 0,C 180,E1 -3768.849,E2 -3768.849} C_VEL
LIN {X 0,Y 545.125,Z 516.58,A -85,B 0,C 180,E1 -3771.847,E2 -3771.847} C_VEL
LIN {X 0,Y 545.2,Z 516.568,A -85,B 0,C 180,E1 -3774.823,E2 -3774.823} C_VEL
LIN {X 0,Y 545.186,Z 516.573,A -85,B 0,C 180,E1 -3777.784,E2 -3777.784} C_VEL
LIN {X 0,Y 545.207,Z 516.567,A -85,B 0,C 180,E1 -3780.739,E2 -3780.739} C_VEL
LIN {X 0,Y 545.169,Z 516.573,A -85,B 0,C 180,E1 -3782.956,E2 -3782.956} C_VEL
LIN {X 0,Y 545.162,Z 516.574,A -85,B 0,C 180,E1 -3785.92,E2 -3785.92} C_VEL
LIN {X 0,Y 545.119,Z 516.579,A -85,B 0,C 180,E1 -3788.9,E2 -3788.9} C_VEL
LIN {X 0,Y 545.126,Z 516.579,A -85,B 0,C 180,E1 -3791.905,E2 -3791.905} C_VEL
LIN {X 0,Y 545.076,Z 516.585,A -85,B 0,C 180,E1 -3794.944,E2 -3794.944} C_VEL
LIN {X 0,Y 545.074,Z 516.584,A -85,B 0,C 180,E1 -3798.026,E2 -3798.026} C_VEL
LIN {X 0,Y 545.09,Z 516.58,A -85,B 0,C 180,E1 -3800.372,E2 -3800.372} C_VEL
LIN {X 0,Y 545.083,Z 516.589,A -85,B 0,C 180,E1 -3803.559,E2 -3803.559} C_VEL
LIN {X 0,Y 545.082,Z 516.583,A -85,B 0,C 180,E1 -3806.001,E2 -3806.001} C_VEL
LIN {X 0,Y 545.086,Z 516.582,A -85,B 0,C 180,E1 -3808.75,E2 -3808.75} C_VEL
LIN {X 0,Y 545.071,Z 516.588,A -85,B 0,C 180,E1 -3811.683,E2 -3811.683} C_VEL
LIN {X 0,Y 545.08,Z 516.582,A -85,B 0,C 180,E1 -3814.564,E2 -3814.564} C_VEL
LIN {X 0,Y 545.059,Z 516.588,A -85,B 0,C 180,E1 -3817.02,E2 -3817.02} C_VEL
LIN {X 0,Y 544.353,Z 516.682,A -85,B 0,C 180,E1 -3817.636,E2 -3817.636} C_VEL
LIN {X 0,Y 541.491,Z 517.038,A -85,B 0,C 180,E1 -3818.637,E2 -3818.637} C_VEL
LIN {X 0,Y 539.106,Z 517.335,A -85,B 0,C 180,E1 -3819.443,E2 -3819.443} C_VEL
LIN {X 0,Y 538.096,Z 517.453,A -85,B 0,C 180,E1 -3820.065,E2 -3820.065} C_VEL
LIN {X 0,Y 538.019,Z 517.461,A -85,B 0,C 180,E1 -3820.276,E2 -3820.276} C_VEL
LIN {X 0,Y 538.027,Z 517.464,A -85,B 0,C 180,E1 -3822.989,E2 -3822.989} C_VEL
LIN {X 0,Y 538.027,Z 517.463,A -85,B 0,C 180,E1 -3825.926,E2 -3825.926} C_VEL
LIN {X 0,Y 538.077,Z 517.461,A -85,B 0,C 180,E1 -3829.25,E2 -3829.25} C_VEL
LIN {X 0,Y 537.993,Z 517.465,A -85,B 0,C 180,E1 -3832.123,E2 -3832.123} C_VEL
LIN {X 0,Y 538.011,Z 517.465,A -85,B 0,C 180,E1 -3834.918,E2 -3834.918} C_VEL
LIN {X 0,Y 538.026,Z 517.467,A -85,B 0,C 180,E1 -3837.619,E2 -3837.619} C_VEL
LIN {X 0,Y 538.018,Z 517.462,A -85,B 0,C 180,E1 -3840.24,E2 -3840.24} C_VEL
LIN {X 0,Y 538.065,Z 517.457,A -85,B 0,C 180,E1 -3842.797,E2 -3842.797} C_VEL
LIN {X 0,Y 538.05,Z 517.466,A -85,B 0,C 180,E1 -3845.293,E2 -3845.293} C_VEL
LIN {X 0,Y 538.025,Z 517.463,A -85,B 0,C 180,E1 -3848.547,E2 -3848.547} C_VEL
LIN {X 0,Y 538.041,Z 517.465,A -85,B 0,C 180,E1 -3850.941,E2 -3850.941} C_VEL
LIN {X 0,Y 538.102,Z 517.545,A -85,B 0,C 180,E1 -3853.692,E2 -3853.692} C_VEL
LIN {X 0,Y 538.706,Z 521.557,A -85,B 0,C 180,E1 -3854.488,E2 -3854.488} C_VEL
LIN {X 0,Y 538.319,Z 538.868,A -85,B 0,C 180,E1 -3857.752,E2 -3857.752} C_VEL
LIN {X 0,Y 538.188,Z 547.177,A -85,B 0,C 180,E1 -3859.3,E2 -3859.3} C_VEL
LIN {X 0,Y 539.698,Z 556.958,A -85,B 0,C 180,E1 -3859.48,E2 -3859.48} C_VEL
LIN {X 0,Y 539.326,Z 653.942,A -85,B 0,C 180,E1 -3860.791,E2 -3860.791} C_VEL
LIN {X 0,Y 539.162,Z 667.1,A -85,B 0,C 180,E1 -3861.119,E2 -3861.119} C_VEL
LIN {X 0,Y 538.953,Z 680.289,A -85,B 0,C 180,E1 -3861.612,E2 -3861.612} C_VEL
LIN {X 0,Y 538.749,Z 692.173,A -85,B 0,C 180,E1 -3862.222,E2 -3862.222} C_VEL
LIN {X 0,Y 538.46,Z 703.634,A -85,B 0,C 180,E1 -3862.978,E2 -3862.978} C_VEL
LIN {X 0,Y 538.312,Z 713.81,A -85,B 0,C 180,E1 -3863.817,E2 -3863.817} C_VEL
LIN {X 0,Y 538.13,Z 723.064,A -85,B 0,C 180,E1 -3864.755,E2 -3864.755} C_VEL
LIN {X 0,Y 537.872,Z 732.033,A -85,B 0,C 180,E1 -3865.879,E2 -3865.879} C_VEL
LIN {X 0,Y 537.685,Z 739.276,A -85,B 0,C 180,E1 -3867.003,E2 -3867.003} C_VEL
LIN {X 0,Y 537.634,Z 745.087,A -85,B 0,C 180,E1 -3868.127,E2 -3868.127} C_VEL
LIN {X 0,Y 537.482,Z 749.68,A -85,B 0,C 180,E1 -3869.251,E2 -3869.251} C_VEL
LIN {X 0,Y 537.484,Z 752.12,A -85,B 0,C 180,E1 -3870,E2 -3870} C_VEL
LIN {X 0,Y 537.449,Z 754.111,A -85,B 0,C 180,E1 -3870.749,E2 -3870.749} C_VEL
LIN {X 0,Y 537.453,Z 755.69,A -85,B 0,C 180,E1 -3871.499,E2 -3871.499} C_VEL
LIN {X 0,Y 537.489,Z 756.861,A -85,B 0,C 180,E1 -3872.248,E2 -3872.248} C_VEL
LIN {X 0,Y 537.545,Z 757.596,A -85,B 0,C 180,E1 -3872.998,E2 -3872.998} C_VEL
LIN {X 0,Y 537.561,Z 757.944,A -85,B 0,C 180,E1 -3873.748,E2 -3873.748} C_VEL
LIN {X 0,Y 537.52,Z 757.486,A -85,B 0,C 180,E1 -3875.251,E2 -3875.251} C_VEL
LIN {X 0,Y 537.537,Z 755.947,A -85,B 0,C 180,E1 -3876.453,E2 -3876.453} C_VEL
LIN {X 0,Y 537.557,Z 752.683,A -85,B 0,C 180,E1 -3877.89,E2 -3877.89} C_VEL
LIN {X 0,Y 537.573,Z 748.971,A -85,B 0,C 180,E1 -3879.026,E2 -3879.026} C_VEL
LIN {X 0,Y 537.649,Z 744.121,A -85,B 0,C 180,E1 -3880.164,E2 -3880.164} C_VEL
LIN {X 0,Y 537.774,Z 737.981,A -85,B 0,C 180,E1 -3881.305,E2 -3881.305} C_VEL
LIN {X 0,Y 537.891,Z 730.32,A -85,B 0,C 180,E1 -3882.45,E2 -3882.45} C_VEL
LIN {X 0,Y 538.085,Z 722.454,A -85,B 0,C 180,E1 -3883.405,E2 -3883.405} C_VEL
LIN {X 0,Y 538.286,Z 712.807,A -85,B 0,C 180,E1 -3884.363,E2 -3884.363} C_VEL
LIN {X 0,Y 538.465,Z 702.061,A -85,B 0,C 180,E1 -3885.228,E2 -3885.228} C_VEL
LIN {X 0,Y 538.723,Z 691.661,A -85,B 0,C 180,E1 -3885.9,E2 -3885.9} C_VEL
LIN {X 0,Y 538.958,Z 679.205,A -85,B 0,C 180,E1 -3886.525,E2 -3886.525} C_VEL
LIN {X 0,Y 539.135,Z 665.993,A -85,B 0,C 180,E1 -3887.007,E2 -3887.007} C_VEL
LIN {X 0,Y 539.318,Z 652.919,A -85,B 0,C 180,E1 -3887.318,E2 -3887.318} C_VEL
LIN {X 0,Y 539.574,Z 555.616,A -85,B 0,C 180,E1 -3888.631,E2 -3888.631} C_VEL
LIN {X 0,Y 538.167,Z 547.096,A -85,B 0,C 180,E1 -3888.808,E2 -3888.808} C_VEL
LIN {X 0,Y 538.466,Z 531.323,A -85,B 0,C 180,E1 -3891.764,E2 -3891.764} C_VEL
LIN {X 0,Y 538.652,Z 521.333,A -85,B 0,C 180,E1 -3893.653,E2 -3893.653} C_VEL
LIN {X 0,Y 538.054,Z 517.467,A -85,B 0,C 180,E1 -3894.453,E2 -3894.453} C_VEL
LIN {X 0,Y 538.059,Z 517.46,A -85,B 0,C 180,E1 -3897.351,E2 -3897.351} C_VEL
LIN {X 0,Y 538.019,Z 517.463,A -85,B 0,C 180,E1 -3899.76,E2 -3899.76} C_VEL
LIN {X 0,Y 538.026,Z 517.466,A -85,B 0,C 180,E1 -3902.381,E2 -3902.381} C_VEL
LIN {X 0,Y 538.012,Z 517.467,A -85,B 0,C 180,E1 -3905.082,E2 -3905.082} C_VEL
LIN {X 0,Y 537.993,Z 517.465,A -85,B 0,C 180,E1 -3907.877,E2 -3907.877} C_VEL
LIN {X 0,Y 538.076,Z 517.463,A -85,B 0,C 180,E1 -3910.772,E2 -3910.772} C_VEL
LIN {X 0,Y 538.027,Z 517.462,A -85,B 0,C 180,E1 -3914.074,E2 -3914.074} C_VEL
LIN {X 0,Y 538.02,Z 517.463,A -85,B 0,C 180,E1 -3917.214,E2 -3917.214} C_VEL
LIN {X 0,Y 538.025,Z 517.462,A -85,B 0,C 180,E1 -3920.203,E2 -3920.203} C_VEL
LIN {X 0,Y 538.025,Z 517.464,A -85,B 0,C 180,E1 -3923.067,E2 -3923.067} C_VEL
LIN {X 0,Y 538.027,Z 517.46,A -85,B 0,C 180,E1 -3925.827,E2 -3925.827} C_VEL
LIN {X 0,Y 538.018,Z 517.469,A -85,B 0,C 180,E1 -3928.499,E2 -3928.499} C_VEL
LIN {X 0,Y 538.052,Z 517.461,A -85,B 0,C 180,E1 -3931.099,E2 -3931.099} C_VEL
LIN {X 0,Y 538.043,Z 517.457,A -85,B 0,C 180,E1 -3933.633,E2 -3933.633} C_VEL
LIN {X 0,Y 538.014,Z 517.465,A -85,B 0,C 180,E1 -3936.117,E2 -3936.117} C_VEL
LIN {X 0,Y 538.034,Z 517.461,A -85,B 0,C 180,E1 -3939.348,E2 -3939.348} C_VEL
LIN {X 0,Y 538.064,Z 517.463,A -85,B 0,C 180,E1 -3942.517,E2 -3942.517} C_VEL
LIN {X 0,Y 538.054,Z 517.457,A -85,B 0,C 180,E1 -3945.63,E2 -3945.63} C_VEL
LIN {X 0,Y 538.08,Z 517.463,A -85,B 0,C 180,E1 -3948.701,E2 -3948.701} C_VEL
LIN {X 0,Y 538.083,Z 517.453,A -85,B 0,C 180,E1 -3951.739,E2 -3951.739} C_VEL
LIN {X 0,Y 538.176,Z 517.45,A -85,B 0,C 180,E1 -3954.755,E2 -3954.755} C_VEL
LIN {X 0,Y 538.158,Z 517.442,A -85,B 0,C 180,E1 -3957.755,E2 -3957.755} C_VEL
LIN {X 0,Y 538.176,Z 517.449,A -85,B 0,C 180,E1 -3960.748,E2 -3960.748} C_VEL
LIN {X 0,Y 538.135,Z 517.449,A -85,B 0,C 180,E1 -3962.994,E2 -3962.994} C_VEL
LIN {X 0,Y 538.115,Z 517.451,A -85,B 0,C 180,E1 -3965.997,E2 -3965.997} C_VEL
LIN {X 0,Y 538.068,Z 517.458,A -85,B 0,C 180,E1 -3969.018,E2 -3969.018} C_VEL
LIN {X 0,Y 538.074,Z 517.457,A -85,B 0,C 180,E1 -3972.063,E2 -3972.063} C_VEL
LIN {X 0,Y 538.036,Z 517.462,A -85,B 0,C 180,E1 -3975.144,E2 -3975.144} C_VEL
LIN {X 0,Y 538.026,Z 517.465,A -85,B 0,C 180,E1 -3978.27,E2 -3978.27} C_VEL
LIN {X 0,Y 538.033,Z 517.469,A -85,B 0,C 180,E1 -3980.652,E2 -3980.652} C_VEL
LIN {X 0,Y 538.015,Z 517.462,A -85,B 0,C 180,E1 -3983.888,E2 -3983.888} C_VEL
LIN {X 0,Y 538.042,Z 517.465,A -85,B 0,C 180,E1 -3986.367,E2 -3986.367} C_VEL
LIN {X 0,Y 538.048,Z 517.462,A -85,B 0,C 180,E1 -3988.939,E2 -3988.939} C_VEL
LIN {X 0,Y 538.02,Z 517.462,A -85,B 0,C 180,E1 -3991.891,E2 -3991.891} C_VEL
LIN {X 0,Y 538.028,Z 517.47,A -85,B 0,C 180,E1 -3994.622,E2 -3994.622} C_VEL
LIN {X 0,Y 538.001,Z 517.465,A -85,B 0,C 180,E1 -3997.171,E2 -3997.171} C_VEL
LIN {X 0,Y 538.049,Z 517.459,A -85,B 0,C 180,E1 -3999.795,E2 -3999.795} C_VEL
LIN {X 0,Y 538.014,Z 517.469,A -85,B 0,C 180,E1 -4002.787,E2 -4002.787} C_VEL
LIN {X 0,Y 538.028,Z 517.463,A -85,B 0,C 180,E1 -4005.141,E2 -4005.141} C_VEL
LIN {X 0,Y 538.038,Z 517.465,A -85,B 0,C 180,E1 -4008.229,E2 -4008.229} C_VEL
LIN {X 0,Y 538.015,Z 517.464,A -85,B 0,C 180,E1 -4011.171,E2 -4011.171} C_VEL
LIN {X 0,Y 537.999,Z 517.468,A -85,B 0,C 180,E1 -4014.088,E2 -4014.088} C_VEL
LIN {X 0,Y 538.03,Z 517.468,A -85,B 0,C 180,E1 -4016.728,E2 -4016.728} C_VEL
LIN {X 0,Y 538.025,Z 517.462,A -85,B 0,C 180,E1 -4019.557,E2 -4019.557} C_VEL
LIN {X 0,Y 538.044,Z 517.462,A -85,B 0,C 180,E1 -4021.951,E2 -4021.951} C_VEL
LIN {X 0,Y 538.072,Z 517.464,A -85,B 0,C 180,E1 -4024.468,E2 -4024.468} C_VEL
LIN {X 0,Y 538.024,Z 517.479,A -85,B 0,C 180,E1 -4026.119,E2 -4026.119} C_VEL
LIN {X 0,Y 539.343,Z 525.375,A -85,B 0,C 180,E1 -4027.434,E2 -4027.434} C_VEL
LIN {X 0,Y 538.916,Z 544.199,A -85,B 0,C 180,E1 -4030.379,E2 -4030.379} C_VEL
LIN {X 0,Y 538.559,Z 562.008,A -85,B 0,C 180,E1 -4033.121,E2 -4033.121} C_VEL
LIN {X 0,Y 538.379,Z 575.998,A -85,B 0,C 180,E1 -4035.251,E2 -4035.251} C_VEL
LIN {X 0,Y 539.676,Z 584.583,A -85,B 0,C 180,E1 -4035.403,E2 -4035.403} C_VEL
LIN {X 0,Y 539.312,Z 683.961,A -85,B 0,C 180,E1 -4036.746,E2 -4036.746} C_VEL
LIN {X 0,Y 539.168,Z 697.227,A -85,B 0,C 180,E1 -4037.078,E2 -4037.078} C_VEL
LIN {X 0,Y 538.971,Z 709.376,A -85,B 0,C 180,E1 -4037.528,E2 -4037.528} C_VEL
LIN {X 0,Y 538.787,Z 720.792,A -85,B 0,C 180,E1 -4038.096,E2 -4038.096} C_VEL
LIN {X 0,Y 538.535,Z 731.906,A -85,B 0,C 180,E1 -4038.807,E2 -4038.807} C_VEL
LIN {X 0,Y 538.266,Z 742.539,A -85,B 0,C 180,E1 -4039.658,E2 -4039.658} C_VEL
LIN {X 0,Y 538.066,Z 752.115,A -85,B 0,C 180,E1 -4040.603,E2 -4040.603} C_VEL
LIN {X 0,Y 537.921,Z 759.962,A -85,B 0,C 180,E1 -4041.548,E2 -4041.548} C_VEL
LIN {X 0,Y 537.754,Z 767.623,A -85,B 0,C 180,E1 -4042.679,E2 -4042.679} C_VEL
LIN {X 0,Y 537.693,Z 774.68,A -85,B 0,C 180,E1 -4043.998,E2 -4043.998} C_VEL
LIN {X 0,Y 537.54,Z 779.373,A -85,B 0,C 180,E1 -4045.125,E2 -4045.125} C_VEL
LIN {X 0,Y 537.591,Z 782.958,A -85,B 0,C 180,E1 -4046.252,E2 -4046.252} C_VEL
LIN {X 0,Y 537.551,Z 784.807,A -85,B 0,C 180,E1 -4047.002,E2 -4047.002} C_VEL
LIN {X 0,Y 537.451,Z 787.183,A -85,B 0,C 180,E1 -4048.501,E2 -4048.501} C_VEL
LIN {X 0,Y 537.442,Z 788,A -85,B 0,C 180,E1 -4050,E2 -4050} C_VEL
LIN {X 0,Y 537.451,Z 787.184,A -85,B 0,C 180,E1 -4051.499,E2 -4051.499} C_VEL
LIN {X 0,Y 537.551,Z 784.81,A -85,B 0,C 180,E1 -4052.998,E2 -4052.998} C_VEL
LIN {X 0,Y 537.603,Z 781.896,A -85,B 0,C 180,E1 -4054.123,E2 -4054.123} C_VEL
LIN {X 0,Y 537.588,Z 777.949,A -85,B 0,C 180,E1 -4055.25,E2 -4055.25} C_VEL
LIN {X 0,Y 537.65,Z 773.081,A -85,B 0,C 180,E1 -4056.335,E2 -4056.335} C_VEL
LIN {X 0,Y 537.79,Z 766.468,A -85,B 0,C 180,E1 -4057.509,E2 -4057.509} C_VEL
LIN {X 0,Y 537.972,Z 758.479,A -85,B 0,C 180,E1 -4058.64,E2 -4058.64} C_VEL
LIN {X 0,Y 538.143,Z 750.336,A -85,B 0,C 180,E1 -4059.585,E2 -4059.585} C_VEL
LIN {X 0,Y 538.352,Z 740.401,A -85,B 0,C 180,E1 -4060.531,E2 -4060.531} C_VEL
LIN {X 0,Y 538.578,Z 730.595,A -85,B 0,C 180,E1 -4061.288,E2 -4061.288} C_VEL
LIN {X 0,Y 538.804,Z 719.707,A -85,B 0,C 180,E1 -4061.963,E2 -4061.963} C_VEL
LIN {X 0,Y 538.991,Z 707.109,A -85,B 0,C 180,E1 -4062.567,E2 -4062.567} C_VEL
LIN {X 0,Y 539.164,Z 694.098,A -85,B 0,C 180,E1 -4063.018,E2 -4063.018} C_VEL
LIN {X 0,Y 539.368,Z 681.124,A -85,B 0,C 180,E1 -4063.3,E2 -4063.3} C_VEL
LIN {X 0,Y 539.577,Z 583.411,A -85,B 0,C 180,E1 -4064.616,E2 -4064.616} C_VEL
LIN {X 0,Y 538.362,Z 575.928,A -85,B 0,C 180,E1 -4064.751,E2 -4064.751} C_VEL
LIN {X 0,Y 538.749,Z 554.103,A -85,B 0,C 180,E1 -4068.089,E2 -4068.089} C_VEL
LIN {X 0,Y 539.128,Z 534.023,A -85,B 0,C 180,E1 -4071.207,E2 -4071.207} C_VEL
LIN {X 0,Y 539.274,Z 523.834,A -85,B 0,C 180,E1 -4072.811,E2 -4072.811} C_VEL
LIN {X 0,Y 538.043,Z 517.467,A -85,B 0,C 180,E1 -4073.886,E2 -4073.886} C_VEL
LIN {X 0,Y 538.042,Z 517.461,A -85,B 0,C 180,E1 -4076.366,E2 -4076.366} C_VEL
LIN {X 0,Y 538.03,Z 517.464,A -85,B 0,C 180,E1 -4078.933,E2 -4078.933} C_VEL
LIN {X 0,Y 538.027,Z 517.464,A -85,B 0,C 180,E1 -4081.89,E2 -4081.89} C_VEL
LIN {X 0,Y 538.024,Z 517.461,A -85,B 0,C 180,E1 -4084.619,E2 -4084.619} C_VEL
LIN {X 0,Y 538.004,Z 517.468,A -85,B 0,C 180,E1 -4087.17,E2 -4087.17} C_VEL
LIN {X 0,Y 538.03,Z 517.465,A -85,B 0,C 180,E1 -4089.795,E2 -4089.795} C_VEL
LIN {X 0,Y 538.02,Z 517.462,A -85,B 0,C 180,E1 -4092.785,E2 -4092.785} C_VEL
LIN {X 0,Y 538.025,Z 517.464,A -85,B 0,C 180,E1 -4095.925,E2 -4095.925} C_VEL
LIN {X 0,Y 538.073,Z 517.461,A -85,B 0,C 180,E1 -4099.248,E2 -4099.248} C_VEL
LIN {X 0,Y 537.988,Z 517.466,A -85,B 0,C 180,E1 -4102.122,E2 -4102.122} C_VEL
LIN {X 0,Y 538.015,Z 517.464,A -85,B 0,C 180,E1 -4104.917,E2 -4104.917} C_VEL
LIN {X 0,Y 538.025,Z 517.468,A -85,B 0,C 180,E1 -4107.618,E2 -4107.618} C_VEL
LIN {X 0,Y 538.036,Z 517.46,A -85,B 0,C 180,E1 -4110.24,E2 -4110.24} C_VEL
LIN {X 0,Y 538.063,Z 517.457,A -85,B 0,C 180,E1 -4112.796,E2 -4112.796} C_VEL
LIN {X 0,Y 538.041,Z 517.466,A -85,B 0,C 180,E1 -4115.292,E2 -4115.292} C_VEL
LIN {X 0,Y 538.006,Z 517.465,A -85,B 0,C 180,E1 -4118.041,E2 -4118.041} C_VEL
LIN {X 0,Y 538.032,Z 517.462,A -85,B 0,C 180,E1 -4120.94,E2 -4120.94} C_VEL
LIN {X 0,Y 538.018,Z 517.469,A -85,B 0,C 180,E1 -4123.299,E2 -4123.299} C_VEL
LIN {X 0,Y 538.054,Z 517.464,A -85,B 0,C 180,E1 -4125.63,E2 -4125.63} C_VEL
LIN {X 0,Y 538.079,Z 517.454,A -85,B 0,C 180,E1 -4128.702,E2 -4128.702} C_VEL
LIN {X 0,Y 538.081,Z 517.458,A -85,B 0,C 180,E1 -4131.74,E2 -4131.74} C_VEL
LIN {X 0,Y 538.157,Z 517.445,A -85,B 0,C 180,E1 -4134.755,E2 -4134.755} C_VEL
LIN {X 0,Y 538.158,Z 517.449,A -85,B 0,C 180,E1 -4137.755,E2 -4137.755} C_VEL
LIN {X 0,Y 538.176,Z 517.443,A -85,B 0,C 180,E1 -4140.748,E2 -4140.748} C_VEL
LIN {X 0,Y 538.135,Z 517.45,A -85,B 0,C 180,E1 -4142.995,E2 -4142.995} C_VEL
LIN {X 0,Y 538.115,Z 517.451,A -85,B 0,C 180,E1 -4145.998,E2 -4145.998} C_VEL
LIN {X 0,Y 538.068,Z 517.459,A -85,B 0,C 180,E1 -4149.018,E2 -4149.018} C_VEL
LIN {X 0,Y 538.074,Z 517.456,A -85,B 0,C 180,E1 -4152.063,E2 -4152.063} C_VEL
LIN {X 0,Y 538.036,Z 517.464,A -85,B 0,C 180,E1 -4155.144,E2 -4155.144} C_VEL
LIN {X 0,Y 538.026,Z 517.461,A -85,B 0,C 180,E1 -4158.271,E2 -4158.271} C_VEL
LIN {X 0,Y 538.034,Z 517.46,A -85,B 0,C 180,E1 -4160.652,E2 -4160.652} C_VEL
LIN {X 0,Y 538.016,Z 517.465,A -85,B 0,C 180,E1 -4163.888,E2 -4163.888} C_VEL
LIN {X 0,Y 538.043,Z 517.458,A -85,B 0,C 180,E1 -4166.367,E2 -4166.367} C_VEL
LIN {X 0,Y 538.049,Z 517.46,A -85,B 0,C 180,E1 -4168.939,E2 -4168.939} C_VEL
LIN {X 0,Y 538.021,Z 517.464,A -85,B 0,C 180,E1 -4171.891,E2 -4171.891} C_VEL
LIN {X 0,Y 538.029,Z 517.46,A -85,B 0,C 180,E1 -4174.622,E2 -4174.622} C_VEL
LIN {X 0,Y 538.003,Z 517.469,A -85,B 0,C 180,E1 -4177.171,E2 -4177.171} C_VEL
LIN {X 0,Y 538.019,Z 517.461,A -85,B 0,C 180,E1 -4180.276,E2 -4180.276} C_VEL
LIN {X 0,Y 537.368,Z 517.546,A -85,B 0,C 180,E1 -4180.901,E2 -4180.901} C_VEL
LIN {X 0,Y 534.517,Z 517.908,A -85,B 0,C 180,E1 -4181.916,E2 -4181.916} C_VEL
LIN {X 0,Y 532.093,Z 518.213,A -85,B 0,C 180,E1 -4182.733,E2 -4182.733} C_VEL
LIN {X 0,Y 531.045,Z 518.34,A -85,B 0,C 180,E1 -4183.364,E2 -4183.364} C_VEL
LIN {X 0,Y 530.957,Z 518.348,A -85,B 0,C 180,E1 -4183.578,E2 -4183.578} C_VEL
LIN {X 0,Y 530.965,Z 518.34,A -85,B 0,C 180,E1 -4186.507,E2 -4186.507} C_VEL
LIN {X 0,Y 531.025,Z 518.339,A -85,B 0,C 180,E1 -4189.572,E2 -4189.572} C_VEL
LIN {X 0,Y 530.967,Z 518.34,A -85,B 0,C 180,E1 -4192.578,E2 -4192.578} C_VEL
LIN {X 0,Y 530.995,Z 518.345,A -85,B 0,C 180,E1 -4195.312,E2 -4195.312} C_VEL
LIN {X 0,Y 530.972,Z 518.341,A -85,B 0,C 180,E1 -4198.033,E2 -4198.033} C_VEL
LIN {X 0,Y 530.99,Z 518.339,A -85,B 0,C 180,E1 -4200.875,E2 -4200.875} C_VEL
LIN {X 0,Y 531.006,Z 518.342,A -85,B 0,C 180,E1 -4203.257,E2 -4203.257} C_VEL
LIN {X 0,Y 530.986,Z 518.339,A -85,B 0,C 180,E1 -4205.962,E2 -4205.962} C_VEL
LIN {X 0,Y 531.003,Z 518.342,A -85,B 0,C 180,E1 -4209.063,E2 -4209.063} C_VEL
LIN {X 0,Y 531.021,Z 518.337,A -85,B 0,C 180,E1 -4212.278,E2 -4212.278} C_VEL
LIN {X 0,Y 531.065,Z 518.5,A -85,B 0,C 180,E1 -4213.569,E2 -4213.569} C_VEL
LIN {X 0,Y 531.729,Z 523.015,A -85,B 0,C 180,E1 -4214.476,E2 -4214.476} C_VEL
LIN {X 0,Y 531.327,Z 540.346,A -85,B 0,C 180,E1 -4217.782,E2 -4217.782} C_VEL
LIN {X 0,Y 531.223,Z 547.446,A -85,B 0,C 180,E1 -4219.109,E2 -4219.109} C_VEL
LIN {X 0,Y 532.816,Z 557.016,A -85,B 0,C 180,E1 -4219.287,E2 -4219.287} C_VEL
LIN {X 0,Y 532.431,Z 654.348,A -85,B 0,C 180,E1 -4220.623,E2 -4220.623} C_VEL
LIN {X 0,Y 532.252,Z 667.391,A -85,B 0,C 180,E1 -4220.955,E2 -4220.955} C_VEL
LIN {X 0,Y 532.019,Z 680.504,A -85,B 0,C 180,E1 -4221.454,E2 -4221.454} C_VEL
LIN {X 0,Y 531.806,Z 691.538,A -85,B 0,C 180,E1 -4222.024,E2 -4222.024} C_VEL
LIN {X 0,Y 531.507,Z 702.441,A -85,B 0,C 180,E1 -4222.741,E2 -4222.741} C_VEL
LIN {X 0,Y 531.326,Z 712.297,A -85,B 0,C 180,E1 -4223.545,E2 -4223.545} C_VEL
LIN {X 0,Y 531.065,Z 721.847,A -85,B 0,C 180,E1 -4224.494,E2 -4224.494} C_VEL
LIN {X 0,Y 530.893,Z 729.685,A -85,B 0,C 180,E1 -4225.444,E2 -4225.444} C_VEL
LIN {X 0,Y 530.717,Z 737.372,A -85,B 0,C 180,E1 -4226.584,E2 -4226.584} C_VEL
LIN {X 0,Y 530.49,Z 743.547,A -85,B 0,C 180,E1 -4227.722,E2 -4227.722} C_VEL
LIN {X 0,Y 530.521,Z 748.461,A -85,B 0,C 180,E1 -4228.861,E2 -4228.861} C_VEL
LIN {X 0,Y 530.385,Z 752.271,A -85,B 0,C 180,E1 -4230,E2 -4230} C_VEL
LIN {X 0,Y 530.351,Z 754.237,A -85,B 0,C 180,E1 -4230.759,E2 -4230.759} C_VEL
LIN {X 0,Y 530.362,Z 755.793,A -85,B 0,C 180,E1 -4231.519,E2 -4231.519} C_VEL
LIN {X 0,Y 530.41,Z 756.922,A -85,B 0,C 180,E1 -4232.278,E2 -4232.278} C_VEL
LIN {X 0,Y 530.479,Z 757.955,A -85,B 0,C 180,E1 -4233.798,E2 -4233.798} C_VEL
LIN {X 0,Y 530.394,Z 757.898,A -85,B 0,C 180,E1 -4234.56,E2 -4234.56} C_VEL
LIN {X 0,Y 530.443,Z 757.436,A -85,B 0,C 180,E1 -4235.321,E2 -4235.321} C_VEL
LIN {X 0,Y 530.469,Z 755.261,A -85,B 0,C 180,E1 -4236.848,E2 -4236.848} C_VEL
LIN {X 0,Y 530.48,Z 752.53,A -85,B 0,C 180,E1 -4237.996,E2 -4237.996} C_VEL
LIN {X 0,Y 530.481,Z 748.766,A -85,B 0,C 180,E1 -4239.147,E2 -4239.147} C_VEL
LIN {X 0,Y 530.575,Z 743.86,A -85,B 0,C 180,E1 -4240.301,E2 -4240.301} C_VEL
LIN {X 0,Y 530.722,Z 737.431,A -85,B 0,C 180,E1 -4241.496,E2 -4241.496} C_VEL
LIN {X 0,Y 530.857,Z 729.908,A -85,B 0,C 180,E1 -4242.617,E2 -4242.617} C_VEL
LIN {X 0,Y 531.031,Z 721.938,A -85,B 0,C 180,E1 -4243.586,E2 -4243.586} C_VEL
LIN {X 0,Y 531.315,Z 712.188,A -85,B 0,C 180,E1 -4244.555,E2 -4244.555} C_VEL
LIN {X 0,Y 531.489,Z 701.323,A -85,B 0,C 180,E1 -4245.433,E2 -4245.433} C_VEL
LIN {X 0,Y 531.794,Z 690.759,A -85,B 0,C 180,E1 -4246.112,E2 -4246.112} C_VEL
LIN {X 0,Y 532.073,Z 677.969,A -85,B 0,C 180,E1 -4246.745,E2 -4246.745} C_VEL
LIN {X 0,Y 532.261,Z 665.098,A -85,B 0,C 180,E1 -4247.208,E2 -4247.208} C_VEL
LIN {X 0,Y 532.416,Z 652.591,A -85,B 0,C 180,E1 -4247.5,E2 -4247.5} C_VEL
LIN {X 0,Y 532.706,Z 556.236,A -85,B 0,C 180,E1 -4248.817,E2 -4248.817} C_VEL
LIN {X 0,Y 531.193,Z 547.368,A -85,B 0,C 180,E1 -4248.989,E2 -4248.989} C_VEL
LIN {X 0,Y 531.511,Z 531.546,A -85,B 0,C 180,E1 -4251.991,E2 -4251.991} C_VEL
LIN {X 0,Y 531.682,Z 522.412,A -85,B 0,C 180,E1 -4253.741,E2 -4253.741} C_VEL
LIN {X 0,Y 531.044,Z 518.34,A -85,B 0,C 180,E1 -4254.585,E2 -4254.585} C_VEL
LIN {X 0,Y 531.017,Z 518.336,A -85,B 0,C 180,E1 -4257.595,E2 -4257.595} C_VEL
LIN {X 0,Y 530.975,Z 518.345,A -85,B 0,C 180,E1 -4260.644,E2 -4260.644} C_VEL
LIN {X 0,Y 530.989,Z 518.339,A -85,B 0,C 180,E1 -4263.772,E2 -4263.772} C_VEL
LIN {X 0,Y 530.965,Z 518.349,A -85,B 0,C 180,E1 -4266.557,E2 -4266.557} C_VEL
LIN {X 0,Y 531.004,Z 518.337,A -85,B 0,C 180,E1 -4269.856,E2 -4269.856} C_VEL
LIN {X 0,Y 530.982,Z 518.344,A -85,B 0,C 180,E1 -4272.455,E2 -4272.455} C_VEL
LIN {X 0,Y 530.984,Z 518.338,A -85,B 0,C 180,E1 -4275.62,E2 -4275.62} C_VEL
LIN {X 0,Y 530.996,Z 518.342,A -85,B 0,C 180,E1 -4278.564,E2 -4278.564} C_VEL
LIN {X 0,Y 530.954,Z 518.342,A -85,B 0,C 180,E1 -4281.529,E2 -4281.529} C_VEL
LIN {X 0,Y 530.977,Z 518.344,A -85,B 0,C 180,E1 -4284.381,E2 -4284.381} C_VEL
LIN {X 0,Y 530.969,Z 518.343,A -85,B 0,C 180,E1 -4287.133,E2 -4287.133} C_VEL
LIN {X 0,Y 530.98,Z 518.337,A -85,B 0,C 180,E1 -4289.803,E2 -4289.803} C_VEL
LIN {X 0,Y 531.01,Z 518.342,A -85,B 0,C 180,E1 -4292.466,E2 -4292.466} C_VEL
LIN {X 0,Y 531,Z 518.341,A -85,B 0,C 180,E1 -4294.942,E2 -4294.942} C_VEL
LIN {X 0,Y 530.963,Z 518.342,A -85,B 0,C 180,E1 -4298.246,E2 -4298.246} C_VEL
LIN {X 0,Y 530.99,Z 518.345,A -85,B 0,C 180,E1 -4300.677,E2 -4300.677} C_VEL
LIN {X 0,Y 530.984,Z 518.341,A -85,B 0,C 180,E1 -4303.071,E2 -4303.071} C_VEL
LIN {X 0,Y 531.009,Z 518.335,A -85,B 0,C 180,E1 -4305.435,E2 -4305.435} C_VEL
LIN {X 0,Y 531.037,Z 518.338,A -85,B 0,C 180,E1 -4308.55,E2 -4308.55} C_VEL
LIN {X 0,Y 531.051,Z 518.328,A -85,B 0,C 180,E1 -4311.629,E2 -4311.629} C_VEL
LIN {X 0,Y 531.131,Z 518.328,A -85,B 0,C 180,E1 -4314.685,E2 -4314.685} C_VEL
LIN {X 0,Y 531.13,Z 518.317,A -85,B 0,C 180,E1 -4317.725,E2 -4317.725} C_VEL
LIN {X 0,Y 531.146,Z 518.325,A -85,B 0,C 180,E1 -4320.758,E2 -4320.758} C_VEL
LIN {X 0,Y 531.101,Z 518.324,A -85,B 0,C 180,E1 -4323.034,E2 -4323.034} C_VEL
LIN {X 0,Y 531.075,Z 518.329,A -85,B 0,C 180,E1 -4326.077,E2 -4326.077} C_VEL
LIN {X 0,Y 531.027,Z 518.334,A -85,B 0,C 180,E1 -4329.138,E2 -4329.138} C_VEL
LIN {X 0,Y 531.031,Z 518.336,A -85,B 0,C 180,E1 -4332.225,E2 -4332.225} C_VEL
LIN {X 0,Y 530.986,Z 518.338,A -85,B 0,C 180,E1 -4335.35,E2 -4335.35} C_VEL
LIN {X 0,Y 531.007,Z 518.334,A -85,B 0,C 180,E1 -4337.723,E2 -4337.723} C_VEL
LIN {X 0,Y 530.993,Z 518.341,A -85,B 0,C 180,E1 -4340.938,E2 -4340.938} C_VEL
LIN {X 0,Y 530.971,Z 518.343,A -85,B 0,C 180,E1 -4344.225,E2 -4344.225} C_VEL
LIN {X 0,Y 531.004,Z 518.341,A -85,B 0,C 180,E1 -4346.744,E2 -4346.744} C_VEL
LIN {X 0,Y 530.993,Z 518.338,A -85,B 0,C 180,E1 -4349.322,E2 -4349.322} C_VEL
LIN {X 0,Y 530.973,Z 518.342,A -85,B 0,C 180,E1 -4352.104,E2 -4352.104} C_VEL
LIN {X 0,Y 530.985,Z 518.343,A -85,B 0,C 180,E1 -4354.855,E2 -4354.855} C_VEL
LIN {X 0,Y 530.96,Z 518.341,A -85,B 0,C 180,E1 -4357.508,E2 -4357.508} C_VEL
LIN {X 0,Y 531.021,Z 518.341,A -85,B 0,C 180,E1 -4360.429,E2 -4360.429} C_VEL
LIN {X 0,Y 530.959,Z 518.342,A -85,B 0,C 180,E1 -4363.495,E2 -4363.495} C_VEL
LIN {X 0,Y 530.963,Z 518.35,A -85,B 0,C 180,E1 -4366.507,E2 -4366.507} C_VEL
LIN {X 0,Y 530.983,Z 518.339,A -85,B 0,C 180,E1 -4369.568,E2 -4369.568} C_VEL
LIN {X 0,Y 530.966,Z 518.349,A -85,B 0,C 180,E1 -4372.578,E2 -4372.578} C_VEL
LIN {X 0,Y 530.993,Z 518.338,A -85,B 0,C 180,E1 -4375.311,E2 -4375.311} C_VEL
LIN {X 0,Y 530.982,Z 518.342,A -85,B 0,C 180,E1 -4378.034,E2 -4378.034} C_VEL
LIN {X 0,Y 530.988,Z 518.343,A -85,B 0,C 180,E1 -4380.875,E2 -4380.875} C_VEL
LIN {X 0,Y 531.004,Z 518.339,A -85,B 0,C 180,E1 -4383.257,E2 -4383.257} C_VEL
LIN {X 0,Y 531.009,Z 518.375,A -85,B 0,C 180,E1 -4385.956,E2 -4385.956} C_VEL
LIN {X 0,Y 532.383,Z 526.212,A -85,B 0,C 180,E1 -4387.287,E2 -4387.287} C_VEL
LIN {X 0,Y 531.973,Z 544.018,A -85,B 0,C 180,E1 -4390.112,E2 -4390.112} C_VEL
LIN {X 0,Y 531.594,Z 561.819,A -85,B 0,C 180,E1 -4392.893,E2 -4392.893} C_VEL
LIN {X 0,Y 531.362,Z 575.745,A -85,B 0,C 180,E1 -4395.044,E2 -4395.044} C_VEL
LIN {X 0,Y 532.799,Z 584.948,A -85,B 0,C 180,E1 -4395.217,E2 -4395.217} C_VEL
LIN {X 0,Y 532.422,Z 683.925,A -85,B 0,C 180,E1 -4396.571,E2 -4396.571} C_VEL
LIN {X 0,Y 532.241,Z 697.207,A -85,B 0,C 180,E1 -4396.907,E2 -4396.907} C_VEL
LIN {X 0,Y 532.05,Z 709.375,A -85,B 0,C 180,E1 -4397.363,E2 -4397.363} C_VEL
LIN {X 0,Y 531.828,Z 720.686,A -85,B 0,C 180,E1 -4397.932,E2 -4397.932} C_VEL
LIN {X 0,Y 531.576,Z 731.905,A -85,B 0,C 180,E1 -4398.658,E2 -4398.658} C_VEL
LIN {X 0,Y 531.27,Z 742.538,A -85,B 0,C 180,E1 -4399.52,E2 -4399.52} C_VEL
LIN {X 0,Y 531.06,Z 752.115,A -85,B 0,C 180,E1 -4400.478,E2 -4400.478} C_VEL
LIN {X 0,Y 530.886,Z 759.962,A -85,B 0,C 180,E1 -4401.435,E2 -4401.435} C_VEL
LIN {X 0,Y 530.684,Z 767.622,A -85,B 0,C 180,E1 -4402.581,E2 -4402.581} C_VEL
LIN {X 0,Y 530.604,Z 774.68,A -85,B 0,C 180,E1 -4403.918,E2 -4403.918} C_VEL
LIN {X 0,Y 530.459,Z 779.373,A -85,B 0,C 180,E1 -4405.06,E2 -4405.06} C_VEL
LIN {X 0,Y 530.516,Z 782.958,A -85,B 0,C 180,E1 -4406.202,E2 -4406.202} C_VEL
LIN {X 0,Y 530.457,Z 784.807,A -85,B 0,C 180,E1 -4406.962,E2 -4406.962} C_VEL
LIN {X 0,Y 530.41,Z 786.194,A -85,B 0,C 180,E1 -4407.722,E2 -4407.722} C_VEL
LIN {X 0,Y 530.344,Z 787.786,A -85,B 0,C 180,E1 -4409.241,E2 -4409.241} C_VEL
LIN {X 0,Y 530.342,Z 788,A -85,B 0,C 180,E1 -4410,E2 -4410} C_VEL
LIN {X 0,Y 530.361,Z 787.184,A -85,B 0,C 180,E1 -4411.519,E2 -4411.519} C_VEL
LIN {X 0,Y 530.41,Z 786.196,A -85,B 0,C 180,E1 -4412.278,E2 -4412.278} C_VEL
LIN {X 0,Y 530.457,Z 784.81,A -85,B 0,C 180,E1 -4413.038,E2 -4413.038} C_VEL
LIN {X 0,Y 530.522,Z 781.896,A -85,B 0,C 180,E1 -4414.178,E2 -4414.178} C_VEL
LIN {X 0,Y 530.525,Z 777.948,A -85,B 0,C 180,E1 -4415.321,E2 -4415.321} C_VEL
LIN {X 0,Y 530.599,Z 772.263,A -85,B 0,C 180,E1 -4416.582,E2 -4416.582} C_VEL
LIN {X 0,Y 530.758,Z 765.236,A -85,B 0,C 180,E1 -4417.8,E2 -4417.8} C_VEL
LIN {X 0,Y 530.93,Z 756.994,A -85,B 0,C 180,E1 -4418.948,E2 -4418.948} C_VEL
LIN {X 0,Y 531.137,Z 748.542,A -85,B 0,C 180,E1 -4419.905,E2 -4419.905} C_VEL
LIN {X 0,Y 531.407,Z 738.094,A -85,B 0,C 180,E1 -4420.863,E2 -4420.863} C_VEL
LIN {X 0,Y 531.646,Z 727.138,A -85,B 0,C 180,E1 -4421.672,E2 -4421.672} C_VEL
LIN {X 0,Y 531.933,Z 716.409,A -85,B 0,C 180,E1 -4422.301,E2 -4422.301} C_VEL
LIN {X 0,Y 532.113,Z 704.766,A -85,B 0,C 180,E1 -4422.829,E2 -4422.829} C_VEL
LIN {X 0,Y 532.295,Z 691.327,A -85,B 0,C 180,E1 -4423.262,E2 -4423.262} C_VEL
LIN {X 0,Y 532.46,Z 678.064,A -85,B 0,C 180,E1 -4423.525,E2 -4423.525} C_VEL
LIN {X 0,Y 532.656,Z 583.871,A -85,B 0,C 180,E1 -4424.802,E2 -4424.802} C_VEL
LIN {X 0,Y 531.332,Z 575.698,A -85,B 0,C 180,E1 -4424.964,E2 -4424.964} C_VEL
LIN {X 0,Y 531.748,Z 555.267,A -85,B 0,C 180,E1 -4428.124,E2 -4428.124} C_VEL
LIN {X 0,Y 532.178,Z 535.119,A -85,B 0,C 180,E1 -4431.294,E2 -4431.294} C_VEL
LIN {X 0,Y 532.379,Z 526.222,A -85,B 0,C 180,E1 -4432.713,E2 -4432.713} C_VEL
LIN {X 0,Y 530.996,Z 518.343,A -85,B 0,C 180,E1 -4434.091,E2 -4434.091} C_VEL
LIN {X 0,Y 531.004,Z 518.339,A -85,B 0,C 180,E1 -4436.743,E2 -4436.743} C_VEL
LIN {X 0,Y 530.982,Z 518.347,A -85,B 0,C 180,E1 -4439.322,E2 -4439.322} C_VEL
LIN {X 0,Y 530.979,Z 518.34,A -85,B 0,C 180,E1 -4442.102,E2 -4442.102} C_VEL
LIN {X 0,Y 530.98,Z 518.34,A -85,B 0,C 180,E1 -4444.852,E2 -4444.852} C_VEL
LIN {X 0,Y 530.964,Z 518.35,A -85,B 0,C 180,E1 -4447.507,E2 -4447.507} C_VEL
LIN {X 0,Y 530.983,Z 518.338,A -85,B 0,C 180,E1 -4450.432,E2 -4450.432} C_VEL
LIN {X 0,Y 530.963,Z 518.35,A -85,B 0,C 180,E1 -4453.493,E2 -4453.493} C_VEL
LIN {X 0,Y 530.959,Z 518.341,A -85,B 0,C 180,E1 -4456.505,E2 -4456.505} C_VEL
LIN {X 0,Y 531.021,Z 518.341,A -85,B 0,C 180,E1 -4459.571,E2 -4459.571} C_VEL
LIN {X 0,Y 530.963,Z 518.34,A -85,B 0,C 180,E1 -4462.576,E2 -4462.576} C_VEL
LIN {X 0,Y 530.998,Z 518.343,A -85,B 0,C 180,E1 -4465.311,E2 -4465.311} C_VEL
LIN {X 0,Y 530.975,Z 518.341,A -85,B 0,C 180,E1 -4468.032,E2 -4468.032} C_VEL
LIN {X 0,Y 530.999,Z 518.337,A -85,B 0,C 180,E1 -4470.87,E2 -4470.87} C_VEL
LIN {X 0,Y 531.004,Z 518.342,A -85,B 0,C 180,E1 -4473.256,E2 -4473.256} C_VEL
LIN {X 0,Y 530.988,Z 518.34,A -85,B 0,C 180,E1 -4475.957,E2 -4475.957} C_VEL
LIN {X 0,Y 530.993,Z 518.34,A -85,B 0,C 180,E1 -4479.062,E2 -4479.062} C_VEL
LIN {X 0,Y 531.007,Z 518.335,A -85,B 0,C 180,E1 -4482.277,E2 -4482.277} C_VEL
LIN {X 0,Y 531.03,Z 518.342,A -85,B 0,C 180,E1 -4485.436,E2 -4485.436} C_VEL
LIN {X 0,Y 531.036,Z 518.331,A -85,B 0,C 180,E1 -4488.55,E2 -4488.55} C_VEL
LIN {X 0,Y 531.05,Z 518.336,A -85,B 0,C 180,E1 -4491.629,E2 -4491.629} C_VEL
LIN {X 0,Y 531.115,Z 518.322,A -85,B 0,C 180,E1 -4494.685,E2 -4494.685} C_VEL
LIN {X 0,Y 531.13,Z 518.325,A -85,B 0,C 180,E1 -4497.725,E2 -4497.725} C_VEL
LIN {X 0,Y 531.146,Z 518.319,A -85,B 0,C 180,E1 -4500.758,E2 -4500.758} C_VEL
LIN {X 0,Y 531.101,Z 518.327,A -85,B 0,C 180,E1 -4503.034,E2 -4503.034} C_VEL
LIN {X 0,Y 531.075,Z 518.328,A -85,B 0,C 180,E1 -4506.077,E2 -4506.077} C_VEL
LIN {X 0,Y 531.027,Z 518.337,A -85,B 0,C 180,E1 -4509.138,E2 -4509.138} C_VEL
LIN {X 0,Y 531.032,Z 518.332,A -85,B 0,C 180,E1 -4512.225,E2 -4512.225} C_VEL
LIN {X 0,Y 530.987,Z 518.346,A -85,B 0,C 180,E1 -4515.35,E2 -4515.35} C_VEL
LIN {X 0,Y 531.008,Z 518.34,A -85,B 0,C 180,E1 -4517.723,E2 -4517.723} C_VEL
LIN {X 0,Y 530.994,Z 518.339,A -85,B 0,C 180,E1 -4520.938,E2 -4520.938} C_VEL
LIN {X 0,Y 530.972,Z 518.34,A -85,B 0,C 180,E1 -4524.225,E2 -4524.225} C_VEL
LIN {X 0,Y 531.005,Z 518.336,A -85,B 0,C 180,E1 -4526.744,E2 -4526.744} C_VEL
LIN {X 0,Y 530.994,Z 518.345,A -85,B 0,C 180,E1 -4529.322,E2 -4529.322} C_VEL
LIN {X 0,Y 530.974,Z 518.34,A -85,B 0,C 180,E1 -4532.104,E2 -4532.104} C_VEL
LIN {X 0,Y 530.986,Z 518.339,A -85,B 0,C 180,E1 -4534.855,E2 -4534.855} C_VEL
LIN {X 0,Y 530.961,Z 518.349,A -85,B 0,C 180,E1 -4537.508,E2 -4537.508} C_VEL
LIN {X 0,Y 530.981,Z 518.338,A -85,B 0,C 180,E1 -4540.433,E2 -4540.433} C_VEL
LIN {X 0,Y 530.965,Z 518.348,A -85,B 0,C 180,E1 -4543.283,E2 -4543.283} C_VEL
LIN {X 0,Y 530.957,Z 518.348,A -85,B 0,C 180,E1 -4543.578,E2 -4543.578} C_VEL
LIN {X 0,Y 530.286,Z 518.427,A -85,B 0,C 180,E1 -4544.211,E2 -4544.211} C_VEL
LIN {X 0,Y 527.44,Z 518.786,A -85,B 0,C 180,E1 -4545.24,E2 -4545.24} C_VEL
LIN {X 0,Y 525.038,Z 519.083,A -85,B 0,C 180,E1 -4546.069,E2 -4546.069} C_VEL
LIN {X 0,Y 524.006,Z 519.209,A -85,B 0,C 180,E1 -4546.708,E2 -4546.708} C_VEL
LIN {X 0,Y 523.921,Z 519.22,A -85,B 0,C 180,E1 -4546.925,E2 -4546.925} C_VEL
LIN {X 0,Y 523.977,Z 519.213,A -85,B 0,C 180,E1 -4549.924,E2 -4549.924} C_VEL
LIN {X 0,Y 523.91,Z 519.221,A -85,B 0,C 180,E1 -4552.869,E2 -4552.869} C_VEL
LIN {X 0,Y 523.94,Z 519.22,A -85,B 0,C 180,E1 -4555.711,E2 -4555.711} C_VEL
LIN {X 0,Y 523.924,Z 519.217,A -85,B 0,C 180,E1 -4558.457,E2 -4558.457} C_VEL
LIN {X 0,Y 523.941,Z 519.22,A -85,B 0,C 180,E1 -4561.126,E2 -4561.126} C_VEL
LIN {X 0,Y 523.986,Z 519.211,A -85,B 0,C 180,E1 -4563.981,E2 -4563.981} C_VEL
LIN {X 0,Y 523.927,Z 519.217,A -85,B 0,C 180,E1 -4566.271,E2 -4566.271} C_VEL
LIN {X 0,Y 523.949,Z 519.218,A -85,B 0,C 180,E1 -4568.767,E2 -4568.767} C_VEL
LIN {X 0,Y 523.956,Z 519.223,A -85,B 0,C 180,E1 -4571.221,E2 -4571.221} C_VEL
LIN {X 0,Y 523.99,Z 519.235,A -85,B 0,C 180,E1 -4573.391,E2 -4573.391} C_VEL
LIN {X 0,Y 524.767,Z 524.526,A -85,B 0,C 180,E1 -4574.464,E2 -4574.464} C_VEL
LIN {X 0,Y 524.33,Z 542.111,A -85,B 0,C 180,E1 -4577.86,E2 -4577.86} C_VEL
LIN {X 0,Y 524.279,Z 547.756,A -85,B 0,C 180,E1 -4578.908,E2 -4578.908} C_VEL
LIN {X 0,Y 525.939,Z 557.721,A -85,B 0,C 180,E1 -4579.096,E2 -4579.096} C_VEL
LIN {X 0,Y 525.519,Z 654.863,A -85,B 0,C 180,E1 -4580.45,E2 -4580.45} C_VEL
LIN {X 0,Y 525.35,Z 667.797,A -85,B 0,C 180,E1 -4580.787,E2 -4580.787} C_VEL
LIN {X 0,Y 525.099,Z 680.851,A -85,B 0,C 180,E1 -4581.292,E2 -4581.292} C_VEL
LIN {X 0,Y 524.845,Z 692.629,A -85,B 0,C 180,E1 -4581.918,E2 -4581.918} C_VEL
LIN {X 0,Y 524.47,Z 704.757,A -85,B 0,C 180,E1 -4582.748,E2 -4582.748} C_VEL
LIN {X 0,Y 524.294,Z 715.129,A -85,B 0,C 180,E1 -4583.651,E2 -4583.651} C_VEL
LIN {X 0,Y 524.047,Z 724.118,A -85,B 0,C 180,E1 -4584.613,E2 -4584.613} C_VEL
LIN {X 0,Y 523.778,Z 732.894,A -85,B 0,C 180,E1 -4585.768,E2 -4585.768} C_VEL
LIN {X 0,Y 523.56,Z 739.963,A -85,B 0,C 180,E1 -4586.922,E2 -4586.922} C_VEL
LIN {X 0,Y 523.486,Z 745.603,A -85,B 0,C 180,E1 -4588.077,E2 -4588.077} C_VEL
LIN {X 0,Y 523.291,Z 750.063,A -85,B 0,C 180,E1 -4589.23,E2 -4589.23} C_VEL
LIN {X 0,Y 523.287,Z 752.423,A -85,B 0,C 180,E1 -4590,E2 -4590} C_VEL
LIN {X 0,Y 523.256,Z 754.364,A -85,B 0,C 180,E1 -4590.77,E2 -4590.77} C_VEL
LIN {X 0,Y 523.276,Z 755.894,A -85,B 0,C 180,E1 -4591.539,E2 -4591.539} C_VEL
LIN {X 0,Y 523.334,Z 756.978,A -85,B 0,C 180,E1 -4592.309,E2 -4592.309} C_VEL
LIN {X 0,Y 523.382,Z 757.966,A -85,B 0,C 180,E1 -4593.85,E2 -4593.85} C_VEL
LIN {X 0,Y 523.302,Z 757.886,A -85,B 0,C 180,E1 -4594.622,E2 -4594.622} C_VEL
LIN {X 0,Y 523.347,Z 757.379,A -85,B 0,C 180,E1 -4595.394,E2 -4595.394} C_VEL
LIN {X 0,Y 523.373,Z 755.156,A -85,B 0,C 180,E1 -4596.941,E2 -4596.941} C_VEL
LIN {X 0,Y 523.388,Z 752.377,A -85,B 0,C 180,E1 -4598.105,E2 -4598.105} C_VEL
LIN {X 0,Y 523.398,Z 748.573,A -85,B 0,C 180,E1 -4599.272,E2 -4599.272} C_VEL
LIN {X 0,Y 523.518,Z 743.639,A -85,B 0,C 180,E1 -4600.441,E2 -4600.441} C_VEL
LIN {X 0,Y 523.675,Z 737.408,A -85,B 0,C 180,E1 -4601.613,E2 -4601.613} C_VEL
LIN {X 0,Y 523.837,Z 729.59,A -85,B 0,C 180,E1 -4602.789,E2 -4602.789} C_VEL
LIN {X 0,Y 524.024,Z 721.569,A -85,B 0,C 180,E1 -4603.771,E2 -4603.771} C_VEL
LIN {X 0,Y 524.345,Z 711.752,A -85,B 0,C 180,E1 -4604.753,E2 -4604.753} C_VEL
LIN {X 0,Y 524.587,Z 700.764,A -85,B 0,C 180,E1 -4605.641,E2 -4605.641} C_VEL
LIN {X 0,Y 524.888,Z 689.95,A -85,B 0,C 180,E1 -4606.33,E2 -4606.33} C_VEL
LIN {X 0,Y 525.167,Z 676.867,A -85,B 0,C 180,E1 -4606.972,E2 -4606.972} C_VEL
LIN {X 0,Y 525.423,Z 664.224,A -85,B 0,C 180,E1 -4607.414,E2 -4607.414} C_VEL
LIN {X 0,Y 525.529,Z 650.833,A -85,B 0,C 180,E1 -4607.712,E2 -4607.712} C_VEL
LIN {X 0,Y 525.838,Z 556.906,A -85,B 0,C 180,E1 -4609.008,E2 -4609.008} C_VEL
LIN {X 0,Y 524.221,Z 547.513,A -85,B 0,C 180,E1 -4609.2,E2 -4609.2} C_VEL
LIN {X 0,Y 524.586,Z 531.348,A -85,B 0,C 180,E1 -4612.31,E2 -4612.31} C_VEL
LIN {X 0,Y 524.577,Z 522.722,A -85,B 0,C 180,E1 -4613.991,E2 -4613.991} C_VEL
LIN {X 0,Y 523.996,Z 519.218,A -85,B 0,C 180,E1 -4614.726,E2 -4614.726} C_VEL
LIN {X 0,Y 523.98,Z 519.213,A -85,B 0,C 180,E1 -4617.718,E2 -4617.718} C_VEL
LIN {X 0,Y 523.945,Z 519.22,A -85,B 0,C 180,E1 -4620.854,E2 -4620.854} C_VEL
LIN {X 0,Y 523.96,Z 519.214,A -85,B 0,C 180,E1 -4623.734,E2 -4623.734} C_VEL
LIN {X 0,Y 523.919,Z 519.224,A -85,B 0,C 180,E1 -4626.403,E2 -4626.403} C_VEL
LIN {X 0,Y 523.93,Z 519.221,A -85,B 0,C 180,E1 -4629.083,E2 -4629.083} C_VEL
LIN {X 0,Y 523.97,Z 519.213,A -85,B 0,C 180,E1 -4631.312,E2 -4631.312} C_VEL
LIN {X 0,Y 523.953,Z 519.223,A -85,B 0,C 180,E1 -4634.691,E2 -4634.691} C_VEL
LIN {X 0,Y 523.953,Z 519.214,A -85,B 0,C 180,E1 -4637.881,E2 -4637.881} C_VEL
LIN {X 0,Y 523.919,Z 519.224,A -85,B 0,C 180,E1 -4640.915,E2 -4640.915} C_VEL
LIN {X 0,Y 523.923,Z 519.218,A -85,B 0,C 180,E1 -4643.827,E2 -4643.827} C_VEL
LIN {X 0,Y 523.938,Z 519.223,A -85,B 0,C 180,E1 -4646.635,E2 -4646.635} C_VEL
LIN {X 0,Y 523.957,Z 519.213,A -85,B 0,C 180,E1 -4649.355,E2 -4649.355} C_VEL
LIN {X 0,Y 523.973,Z 519.216,A -85,B 0,C 180,E1 -4652.28,E2 -4652.28} C_VEL
LIN {X 0,Y 523.948,Z 519.221,A -85,B 0,C 180,E1 -4654.581,E2 -4654.581} C_VEL
LIN {X 0,Y 523.909,Z 519.22,A -85,B 0,C 180,E1 -4657.106,E2 -4657.106} C_VEL
LIN {X 0,Y 523.97,Z 519.212,A -85,B 0,C 180,E1 -4659.865,E2 -4659.865} C_VEL
LIN {X 0,Y 523.962,Z 519.219,A -85,B 0,C 180,E1 -4662.837,E2 -4662.837} C_VEL
LIN {X 0,Y 523.967,Z 519.214,A -85,B 0,C 180,E1 -4665.235,E2 -4665.235} C_VEL
LIN {X 0,Y 524.002,Z 519.211,A -85,B 0,C 180,E1 -4668.394,E2 -4668.394} C_VEL
LIN {X 0,Y 523.999,Z 519.207,A -85,B 0,C 180,E1 -4671.516,E2 -4671.516} C_VEL
LIN {X 0,Y 524.09,Z 519.206,A -85,B 0,C 180,E1 -4674.614,E2 -4674.614} C_VEL
LIN {X 0,Y 524.103,Z 519.193,A -85,B 0,C 180,E1 -4677.694,E2 -4677.694} C_VEL
LIN {X 0,Y 524.116,Z 519.2,A -85,B 0,C 180,E1 -4680.768,E2 -4680.768} C_VEL
LIN {X 0,Y 524.067,Z 519.2,A -85,B 0,C 180,E1 -4683.075,E2 -4683.075} C_VEL
LIN {X 0,Y 524.037,Z 519.207,A -85,B 0,C 180,E1 -4686.159,E2 -4686.159} C_VEL
LIN {X 0,Y 523.994,Z 519.209,A -85,B 0,C 180,E1 -4689.262,E2 -4689.262} C_VEL
LIN {X 0,Y 523.998,Z 519.208,A -85,B 0,C 180,E1 -4691.743,E2 -4691.743} C_VEL
LIN {X 0,Y 523.983,Z 519.213,A -85,B 0,C 180,E1 -4695.053,E2 -4695.053} C_VEL
LIN {X 0,Y 523.955,Z 519.214,A -85,B 0,C 180,E1 -4697.969,E2 -4697.969} C_VEL
LIN {X 0,Y 523.963,Z 519.219,A -85,B 0,C 180,E1 -4700.41,E2 -4700.41} C_VEL
LIN {X 0,Y 523.908,Z 519.223,A -85,B 0,C 180,E1 -4702.894,E2 -4702.894} C_VEL
LIN {X 0,Y 523.946,Z 519.215,A -85,B 0,C 180,E1 -4705.419,E2 -4705.419} C_VEL
LIN {X 0,Y 523.963,Z 519.213,A -85,B 0,C 180,E1 -4707.999,E2 -4707.999} C_VEL
LIN {X 0,Y 523.945,Z 519.22,A -85,B 0,C 180,E1 -4710.857,E2 -4710.857} C_VEL
LIN {X 0,Y 523.956,Z 519.214,A -85,B 0,C 180,E1 -4713.736,E2 -4713.736} C_VEL
LIN {X 0,Y 523.916,Z 519.226,A -85,B 0,C 180,E1 -4716.405,E2 -4716.405} C_VEL
LIN {X 0,Y 523.926,Z 519.22,A -85,B 0,C 180,E1 -4719.084,E2 -4719.084} C_VEL
LIN {X 0,Y 523.967,Z 519.213,A -85,B 0,C 180,E1 -4721.313,E2 -4721.313} C_VEL
LIN {X 0,Y 523.951,Z 519.222,A -85,B 0,C 180,E1 -4724.692,E2 -4724.692} C_VEL
LIN {X 0,Y 523.954,Z 519.216,A -85,B 0,C 180,E1 -4727.883,E2 -4727.883} C_VEL
LIN {X 0,Y 523.923,Z 519.222,A -85,B 0,C 180,E1 -4730.917,E2 -4730.917} C_VEL
LIN {X 0,Y 523.903,Z 519.222,A -85,B 0,C 180,E1 -4733.827,E2 -4733.827} C_VEL
LIN {X 0,Y 523.941,Z 519.224,A -85,B 0,C 180,E1 -4736.637,E2 -4736.637} C_VEL
LIN {X 0,Y 523.956,Z 519.215,A -85,B 0,C 180,E1 -4739.357,E2 -4739.357} C_VEL
LIN {X 0,Y 523.978,Z 519.218,A -85,B 0,C 180,E1 -4742.282,E2 -4742.282} C_VEL
LIN {X 0,Y 523.954,Z 519.223,A -85,B 0,C 180,E1 -4744.582,E2 -4744.582} C_VEL
LIN {X 0,Y 523.966,Z 519.315,A -85,B 0,C 180,E1 -4745.796,E2 -4745.796} C_VEL
LIN {X 0,Y 525.422,Z 527.321,A -85,B 0,C 180,E1 -4747.177,E2 -4747.177} C_VEL
LIN {X 0,Y 525.004,Z 545.107,A -85,B 0,C 180,E1 -4750.041,E2 -4750.041} C_VEL
LIN {X 0,Y 524.564,Z 562.901,A -85,B 0,C 180,E1 -4752.858,E2 -4752.858} C_VEL
LIN {X 0,Y 524.32,Z 575.59,A -85,B 0,C 180,E1 -4754.845,E2 -4754.845} C_VEL
LIN {X 0,Y 525.937,Z 585.785,A -85,B 0,C 180,E1 -4755.034,E2 -4755.034} C_VEL
LIN {X 0,Y 525.531,Z 683.712,A -85,B 0,C 180,E1 -4756.392,E2 -4756.392} C_VEL
LIN {X 0,Y 525.311,Z 696.995,A -85,B 0,C 180,E1 -4756.731,E2 -4756.731} C_VEL
LIN {X 0,Y 525.115,Z 709.169,A -85,B 0,C 180,E1 -4757.193,E2 -4757.193} C_VEL
LIN {X 0,Y 524.874,Z 719.832,A -85,B 0,C 180,E1 -4757.732,E2 -4757.732} C_VEL
LIN {X 0,Y 524.649,Z 730.447,A -85,B 0,C 180,E1 -4758.409,E2 -4758.409} C_VEL
LIN {X 0,Y 524.312,Z 741.359,A -85,B 0,C 180,E1 -4759.282,E2 -4759.282} C_VEL
LIN {X 0,Y 524.076,Z 750.26,A -85,B 0,C 180,E1 -4760.155,E2 -4760.155} C_VEL
LIN {X 0,Y 523.851,Z 759.932,A -85,B 0,C 180,E1 -4761.319,E2 -4761.319} C_VEL
LIN {X 0,Y 523.633,Z 767.622,A -85,B 0,C 180,E1 -4762.481,E2 -4762.481} C_VEL
LIN {X 0,Y 523.515,Z 774.68,A -85,B 0,C 180,E1 -4763.835,E2 -4763.835} C_VEL
LIN {X 0,Y 523.384,Z 779.373,A -85,B 0,C 180,E1 -4764.993,E2 -4764.993} C_VEL
LIN {X 0,Y 523.443,Z 782.958,A -85,B 0,C 180,E1 -4766.151,E2 -4766.151} C_VEL
LIN {X 0,Y 523.367,Z 784.807,A -85,B 0,C 180,E1 -4766.921,E2 -4766.921} C_VEL
LIN {X 0,Y 523.334,Z 786.193,A -85,B 0,C 180,E1 -4767.691,E2 -4767.691} C_VEL
LIN {X 0,Y 523.25,Z 787.785,A -85,B 0,C 180,E1 -4769.23,E2 -4769.23} C_VEL
LIN {X 0,Y 523.246,Z 788,A -85,B 0,C 180,E1 -4770,E2 -4770} C_VEL
LIN {X 0,Y 523.274,Z 787.183,A -85,B 0,C 180,E1 -4771.539,E2 -4771.539} C_VEL
LIN {X 0,Y 523.334,Z 786.196,A -85,B 0,C 180,E1 -4772.309,E2 -4772.309} C_VEL
LIN {X 0,Y 523.367,Z 784.81,A -85,B 0,C 180,E1 -4773.079,E2 -4773.079} C_VEL
LIN {X 0,Y 523.441,Z 781.895,A -85,B 0,C 180,E1 -4774.235,E2 -4774.235} C_VEL
LIN {X 0,Y 523.464,Z 777.948,A -85,B 0,C 180,E1 -4775.393,E2 -4775.393} C_VEL
LIN {X 0,Y 523.523,Z 772.727,A -85,B 0,C 180,E1 -4776.581,E2 -4776.581} C_VEL
LIN {X 0,Y 523.665,Z 766.466,A -85,B 0,C 180,E1 -4777.713,E2 -4777.713} C_VEL
LIN {X 0,Y 523.854,Z 758.441,A -85,B 0,C 180,E1 -4778.875,E2 -4778.875} C_VEL
LIN {X 0,Y 524.077,Z 750.261,A -85,B 0,C 180,E1 -4779.845,E2 -4779.845} C_VEL
LIN {X 0,Y 524.354,Z 740.287,A -85,B 0,C 180,E1 -4780.815,E2 -4780.815} C_VEL
LIN {X 0,Y 524.64,Z 728.935,A -85,B 0,C 180,E1 -4781.696,E2 -4781.696} C_VEL
LIN {X 0,Y 524.922,Z 717.994,A -85,B 0,C 180,E1 -4782.369,E2 -4782.369} C_VEL
LIN {X 0,Y 525.158,Z 705.768,A -85,B 0,C 180,E1 -4782.953,E2 -4782.953} C_VEL
LIN {X 0,Y 525.357,Z 692.95,A -85,B 0,C 180,E1 -4783.391,E2 -4783.391} C_VEL
LIN {X 0,Y 525.56,Z 679.368,A -85,B 0,C 180,E1 -4783.681,E2 -4783.681} C_VEL
LIN {X 0,Y 525.849,Z 584.939,A -85,B 0,C 180,E1 -4784.98,E2 -4784.98} C_VEL
LIN {X 0,Y 524.309,Z 575.535,A -85,B 0,C 180,E1 -4785.165,E2 -4785.165} C_VEL
LIN {X 0,Y 524.77,Z 555.521,A -85,B 0,C 180,E1 -4788.303,E2 -4788.303} C_VEL
LIN {X 0,Y 525.239,Z 536.218,A -85,B 0,C 180,E1 -4791.384,E2 -4791.384} C_VEL
LIN {X 0,Y 525.423,Z 527.338,A -85,B 0,C 180,E1 -4792.823,E2 -4792.823} C_VEL
LIN {X 0,Y 523.955,Z 519.22,A -85,B 0,C 180,E1 -4794.23,E2 -4794.23} C_VEL
LIN {X 0,Y 523.952,Z 519.22,A -85,B 0,C 180,E1 -4797.132,E2 -4797.132} C_VEL
LIN {X 0,Y 523.942,Z 519.222,A -85,B 0,C 180,E1 -4799.755,E2 -4799.755} C_VEL
LIN {X 0,Y 523.939,Z 519.215,A -85,B 0,C 180,E1 -4802.448,E2 -4802.448} C_VEL
LIN {X 0,Y 523.925,Z 519.223,A -85,B 0,C 180,E1 -4805.225,E2 -4805.225} C_VEL
LIN {X 0,Y 523.915,Z 519.22,A -85,B 0,C 180,E1 -4808.101,E2 -4808.101} C_VEL
LIN {X 0,Y 523.958,Z 519.22,A -85,B 0,C 180,E1 -4811.31,E2 -4811.31} C_VEL
LIN {X 0,Y 523.951,Z 519.214,A -85,B 0,C 180,E1 -4814.691,E2 -4814.691} C_VEL
